QRS_NEXT_CUT()
PTP {E1 35817.199,E2 35817.199}
PTP {X 0,Y 759.903,A -85,B 0,C 180,E1 35817.199,E2 35817.199,E3 0,E4 0,E5 0,E6 0}
QRS_SPEED_INIT()
LIN {X 0,Y 759.903,Z 1215,A -85,B 0,C 180,E1 35817.199,E2 35817.199,E3 0,E4 0,E5 0,E6 0} C_VEL
LIN {X 0,Y 759.903,Z 294.644,A -85,B 0,C 180,E1 35817.199,E2 35817.199} C_VEL
LIN {X 0,Y 759.903,Z 286.569,A -85,B 0,C 180,E1 35817.199,E2 35817.199} C_VEL
LIN {X 0,Y 759.899,Z 284.569,A -85,B 0,C 180,E1 35817.048,E2 35817.048} C_VEL
LIN {X 0,Y 759.89,Z 284.574,A -85,B 0,C 180,E1 35814.261,E2 35814.261} C_VEL
LIN {X 0,Y 759.904,Z 284.564,A -85,B 0,C 180,E1 35811.373,E2 35811.373} C_VEL
LIN {X 0,Y 759.907,Z 284.576,A -85,B 0,C 180,E1 35808.309,E2 35808.309} C_VEL
LIN {X 0,Y 759.882,Z 284.567,A -85,B 0,C 180,E1 35805.444,E2 35805.444} C_VEL
LIN {X 0,Y 759.904,Z 284.571,A -85,B 0,C 180,E1 35802.621,E2 35802.621} C_VEL
LIN {X 0,Y 759.877,Z 284.573,A -85,B 0,C 180,E1 35799.833,E2 35799.833} C_VEL
LIN {X 0,Y 759.891,Z 284.566,A -85,B 0,C 180,E1 35797.077,E2 35797.077} C_VEL
LIN {X 0,Y 759.911,Z 284.577,A -85,B 0,C 180,E1 35794.097,E2 35794.097} C_VEL
LIN {X 0,Y 759.864,Z 284.571,A -85,B 0,C 180,E1 35791.362,E2 35791.362} C_VEL
LIN {X 0,Y 759.918,Z 284.564,A -85,B 0,C 180,E1 35788.597,E2 35788.597} C_VEL
LIN {X 0,Y 759.88,Z 284.575,A -85,B 0,C 180,E1 35785.632,E2 35785.632} C_VEL
LIN {X 0,Y 759.866,Z 284.568,A -85,B 0,C 180,E1 35782.938,E2 35782.938} C_VEL
LIN {X 0,Y 759.91,Z 284.572,A -85,B 0,C 180,E1 35780.093,E2 35780.093} C_VEL
LIN {X 0,Y 759.867,Z 284.574,A -85,B 0,C 180,E1 35777.337,E2 35777.337} C_VEL
LIN {X 0,Y 759.862,Z 284.57,A -85,B 0,C 180,E1 35774.718,E2 35774.718} C_VEL
LIN {X 0,Y 759.912,Z 284.571,A -85,B 0,C 180,E1 35771.944,E2 35771.944} C_VEL
LIN {X 0,Y 759.864,Z 284.575,A -85,B 0,C 180,E1 35769.168,E2 35769.168} C_VEL
LIN {X 0,Y 759.853,Z 284.57,A -85,B 0,C 180,E1 35766.59,E2 35766.59} C_VEL
LIN {X 0,Y 759.915,Z 284.571,A -85,B 0,C 180,E1 35763.818,E2 35763.818} C_VEL
LIN {X 0,Y 759.913,Z 284.828,A -85,B 0,C 180,E1 35761.644,E2 35761.644} C_VEL
LIN {X 0,Y 759.919,Z 312.056,A -85,B 0,C 180,E1 35759.876,E2 35759.876} C_VEL
LIN {X 0,Y 759.918,Z 346.9,A -85,B 0,C 180,E1 35757.717,E2 35757.717} C_VEL
LIN {X 0,Y 759.914,Z 568.445,A -85,B 0,C 180,E1 35755.191,E2 35755.191} C_VEL
LIN {X 0,Y 759.916,Z 778.609,A -85,B 0,C 180,E1 35752.849,E2 35752.849} C_VEL
LIN {X 0,Y 759.918,Z 798.366,A -85,B 0,C 180,E1 35752.545,E2 35752.545} C_VEL
LIN {X 0,Y 759.911,Z 822.306,A -85,B 0,C 180,E1 35752.064,E2 35752.064} C_VEL
LIN {X 0,Y 759.913,Z 846.929,A -85,B 0,C 180,E1 35751.415,E2 35751.415} C_VEL
LIN {X 0,Y 759.914,Z 866.189,A -85,B 0,C 180,E1 35750.809,E2 35750.809} C_VEL
LIN {X 0,Y 759.917,Z 885.052,A -85,B 0,C 180,E1 35750.125,E2 35750.125} C_VEL
LIN {X 0,Y 759.915,Z 904.461,A -85,B 0,C 180,E1 35749.324,E2 35749.324} C_VEL
LIN {X 0,Y 759.91,Z 928.8,A -85,B 0,C 180,E1 35748.17,E2 35748.17} C_VEL
LIN {X 0,Y 759.915,Z 948.392,A -85,B 0,C 180,E1 35747.102,E2 35747.102} C_VEL
LIN {X 0,Y 759.904,Z 967.176,A -85,B 0,C 180,E1 35745.962,E2 35745.962} C_VEL
LIN {X 0,Y 759.915,Z 988.802,A -85,B 0,C 180,E1 35744.477,E2 35744.477} C_VEL
LIN {X 0,Y 759.916,Z 1005.718,A -85,B 0,C 180,E1 35743.172,E2 35743.172} C_VEL
LIN {X 0,Y 759.903,Z 1024.655,A -85,B 0,C 180,E1 35741.537,E2 35741.537} C_VEL
LIN {X 0,Y 759.903,Z 1039.602,A -85,B 0,C 180,E1 35740.078,E2 35740.078} C_VEL
LIN {X 0,Y 759.901,Z 1054.389,A -85,B 0,C 180,E1 35738.474,E2 35738.474} C_VEL
LIN {X 0,Y 759.889,Z 1068.45,A -85,B 0,C 180,E1 35736.725,E2 35736.725} C_VEL
LIN {X 0,Y 759.91,Z 1079.205,A -85,B 0,C 180,E1 35735.209,E2 35735.209} C_VEL
LIN {X 0,Y 759.908,Z 1089.153,A -85,B 0,C 180,E1 35733.621,E2 35733.621} C_VEL
LIN {X 0,Y 759.901,Z 1099.607,A -85,B 0,C 180,E1 35731.659,E2 35731.659} C_VEL
LIN {X 0,Y 759.92,Z 1106.921,A -85,B 0,C 180,E1 35730,E2 35730} C_VEL
LIN {X 0,Y 759.904,Z 1112.724,A -85,B 0,C 180,E1 35728.417,E2 35728.417} C_VEL
LIN {X 0,Y 759.898,Z 1117.808,A -85,B 0,C 180,E1 35726.681,E2 35726.681} C_VEL
LIN {X 0,Y 759.903,Z 1121.967,A -85,B 0,C 180,E1 35724.64,E2 35724.64} C_VEL
LIN {X 0,Y 759.898,Z 1123.954,A -85,B 0,C 180,E1 35723.047,E2 35723.047} C_VEL
LIN {X 0,Y 759.902,Z 1124.86,A -85,B 0,C 180,E1 35721.449,E2 35721.449} C_VEL
LIN {X 0,Y 759.901,Z 1124.556,A -85,B 0,C 180,E1 35719.538,E2 35719.538} C_VEL
LIN {X 0,Y 759.916,Z 1122.598,A -85,B 0,C 180,E1 35717.693,E2 35717.693} C_VEL
LIN {X 0,Y 759.891,Z 1119.867,A -85,B 0,C 180,E1 35716.144,E2 35716.144} C_VEL
LIN {X 0,Y 759.916,Z 1116.057,A -85,B 0,C 180,E1 35714.587,E2 35714.587} C_VEL
LIN {X 0,Y 759.902,Z 1110.065,A -85,B 0,C 180,E1 35712.701,E2 35712.701} C_VEL
LIN {X 0,Y 759.909,Z 1102.135,A -85,B 0,C 180,E1 35710.796,E2 35710.796} C_VEL
LIN {X 0,Y 759.904,Z 1094.597,A -85,B 0,C 180,E1 35709.271,E2 35709.271} C_VEL
LIN {X 0,Y 759.901,Z 1085.453,A -85,B 0,C 180,E1 35707.672,E2 35707.672} C_VEL
LIN {X 0,Y 759.916,Z 1072.728,A -85,B 0,C 180,E1 35705.762,E2 35705.762} C_VEL
LIN {X 0,Y 759.909,Z 1060.564,A -85,B 0,C 180,E1 35704.182,E2 35704.182} C_VEL
LIN {X 0,Y 759.913,Z 1047.302,A -85,B 0,C 180,E1 35702.644,E2 35702.644} C_VEL
LIN {X 0,Y 759.908,Z 1029.889,A -85,B 0,C 180,E1 35700.867,E2 35700.867} C_VEL
LIN {X 0,Y 759.914,Z 1014.558,A -85,B 0,C 180,E1 35699.477,E2 35699.477} C_VEL
LIN {X 0,Y 759.914,Z 994.945,A -85,B 0,C 180,E1 35697.889,E2 35697.889} C_VEL
LIN {X 0,Y 759.9,Z 977.479,A -85,B 0,C 180,E1 35696.633,E2 35696.633} C_VEL
LIN {X 0,Y 759.915,Z 957.247,A -85,B 0,C 180,E1 35695.323,E2 35695.323} C_VEL
LIN {X 0,Y 759.914,Z 935.774,A -85,B 0,C 180,E1 35694.108,E2 35694.108} C_VEL
LIN {X 0,Y 759.912,Z 917.354,A -85,B 0,C 180,E1 35693.178,E2 35693.178} C_VEL
LIN {X 0,Y 759.915,Z 897.341,A -85,B 0,C 180,E1 35692.279,E2 35692.279} C_VEL
LIN {X 0,Y 759.918,Z 871.571,A -85,B 0,C 180,E1 35691.285,E2 35691.285} C_VEL
LIN {X 0,Y 759.915,Z 851.793,A -85,B 0,C 180,E1 35690.64,E2 35690.64} C_VEL
LIN {X 0,Y 759.916,Z 833.306,A -85,B 0,C 180,E1 35690.123,E2 35690.123} C_VEL
LIN {X 0,Y 759.913,Z 814.474,A -85,B 0,C 180,E1 35689.679,E2 35689.679} C_VEL
LIN {X 0,Y 759.912,Z 795.76,A -85,B 0,C 180,E1 35689.32,E2 35689.32} C_VEL
LIN {X 0,Y 759.913,Z 776.865,A -85,B 0,C 180,E1 35689.038,E2 35689.038} C_VEL
LIN {X 0,Y 759.915,Z 516.196,A -85,B 0,C 180,E1 35686.131,E2 35686.131} C_VEL
LIN {X 0,Y 759.913,Z 346.704,A -85,B 0,C 180,E1 35684.186,E2 35684.186} C_VEL
LIN {X 0,Y 759.917,Z 302.71,A -85,B 0,C 180,E1 35681.441,E2 35681.441} C_VEL
LIN {X 0,Y 759.904,Z 284.847,A -85,B 0,C 180,E1 35680.268,E2 35680.268} C_VEL
LIN {X 0,Y 759.912,Z 284.571,A -85,B 0,C 180,E1 35678.49,E2 35678.49} C_VEL
LIN {X 0,Y 759.917,Z 284.563,A -85,B 0,C 180,E1 35675.467,E2 35675.467} C_VEL
LIN {X 0,Y 759.891,Z 284.574,A -85,B 0,C 180,E1 35672.56,E2 35672.56} C_VEL
LIN {X 0,Y 759.894,Z 284.569,A -85,B 0,C 180,E1 35669.725,E2 35669.725} C_VEL
LIN {X 0,Y 759.894,Z 284.566,A -85,B 0,C 180,E1 35666.998,E2 35666.998} C_VEL
LIN {X 0,Y 759.912,Z 284.578,A -85,B 0,C 180,E1 35664.073,E2 35664.073} C_VEL
LIN {X 0,Y 759.916,Z 284.562,A -85,B 0,C 180,E1 35661.052,E2 35661.052} C_VEL
LIN {X 0,Y 759.911,Z 284.577,A -85,B 0,C 180,E1 35658.012,E2 35658.012} C_VEL
LIN {X 0,Y 759.909,Z 284.564,A -85,B 0,C 180,E1 35655.023,E2 35655.023} C_VEL
LIN {X 0,Y 759.891,Z 284.572,A -85,B 0,C 180,E1 35652.141,E2 35652.141} C_VEL
LIN {X 0,Y 759.894,Z 284.572,A -85,B 0,C 180,E1 35649.391,E2 35649.391} C_VEL
LIN {X 0,Y 759.908,Z 284.563,A -85,B 0,C 180,E1 35646.573,E2 35646.573} C_VEL
LIN {X 0,Y 759.915,Z 284.577,A -85,B 0,C 180,E1 35643.621,E2 35643.621} C_VEL
LIN {X 0,Y 759.907,Z 284.563,A -85,B 0,C 180,E1 35640.603,E2 35640.603} C_VEL
LIN {X 0,Y 759.9,Z 284.574,A -85,B 0,C 180,E1 35637.662,E2 35637.662} C_VEL
LIN {X 0,Y 759.888,Z 284.57,A -85,B 0,C 180,E1 35634.866,E2 35634.866} C_VEL
LIN {X 0,Y 759.9,Z 284.566,A -85,B 0,C 180,E1 35632.059,E2 35632.059} C_VEL
LIN {X 0,Y 759.909,Z 284.576,A -85,B 0,C 180,E1 35629.155,E2 35629.155} C_VEL
LIN {X 0,Y 759.911,Z 284.563,A -85,B 0,C 180,E1 35626.144,E2 35626.144} C_VEL
LIN {X 0,Y 759.919,Z 284.577,A -85,B 0,C 180,E1 35623.095,E2 35623.095} C_VEL
LIN {X 0,Y 759.905,Z 284.563,A -85,B 0,C 180,E1 35620.075,E2 35620.075} C_VEL
LIN {X 0,Y 759.909,Z 284.576,A -85,B 0,C 180,E1 35617.077,E2 35617.077} C_VEL
LIN {X 0,Y 759.883,Z 284.569,A -85,B 0,C 180,E1 35614.264,E2 35614.264} C_VEL
LIN {X 0,Y 759.901,Z 284.566,A -85,B 0,C 180,E1 35611.468,E2 35611.468} C_VEL
LIN {X 0,Y 759.901,Z 284.576,A -85,B 0,C 180,E1 35608.596,E2 35608.596} C_VEL
LIN {X 0,Y 759.899,Z 284.565,A -85,B 0,C 180,E1 35605.721,E2 35605.721} C_VEL
LIN {X 0,Y 759.902,Z 284.574,A -85,B 0,C 180,E1 35602.846,E2 35602.846} C_VEL
LIN {X 0,Y 759.879,Z 284.572,A -85,B 0,C 180,E1 35600.048,E2 35600.048} C_VEL
LIN {X 0,Y 759.91,Z 284.562,A -85,B 0,C 180,E1 35597.238,E2 35597.238} C_VEL
LIN {X 0,Y 759.902,Z 284.796,A -85,B 0,C 180,E1 35594.679,E2 35594.679} C_VEL
LIN {X 0,Y 759.918,Z 288.931,A -85,B 0,C 180,E1 35594.4,E2 35594.4} C_VEL
LIN {X 0,Y 759.896,Z 333.48,A -85,B 0,C 180,E1 35591.844,E2 35591.844} C_VEL
LIN {X 0,Y 759.909,Z 350.22,A -85,B 0,C 180,E1 35590.926,E2 35590.926} C_VEL
LIN {X 0,Y 759.918,Z 558.925,A -85,B 0,C 180,E1 35588.412,E2 35588.412} C_VEL
LIN {X 0,Y 759.917,Z 786.633,A -85,B 0,C 180,E1 35585.769,E2 35585.769} C_VEL
LIN {X 0,Y 759.91,Z 830.472,A -85,B 0,C 180,E1 35585.243,E2 35585.243} C_VEL
LIN {X 0,Y 759.91,Z 856.594,A -85,B 0,C 180,E1 35584.789,E2 35584.789} C_VEL
LIN {X 0,Y 759.914,Z 883.601,A -85,B 0,C 180,E1 35584.163,E2 35584.163} C_VEL
LIN {X 0,Y 759.908,Z 907.506,A -85,B 0,C 180,E1 35583.465,E2 35583.465} C_VEL
LIN {X 0,Y 759.918,Z 931.763,A -85,B 0,C 180,E1 35582.637,E2 35582.637} C_VEL
LIN {X 0,Y 759.917,Z 956.965,A -85,B 0,C 180,E1 35581.611,E2 35581.611} C_VEL
LIN {X 0,Y 759.912,Z 976.742,A -85,B 0,C 180,E1 35580.698,E2 35580.698} C_VEL
LIN {X 0,Y 759.913,Z 995.424,A -85,B 0,C 180,E1 35579.738,E2 35579.738} C_VEL
LIN {X 0,Y 759.909,Z 1013.705,A -85,B 0,C 180,E1 35578.702,E2 35578.702} C_VEL
LIN {X 0,Y 759.911,Z 1035.513,A -85,B 0,C 180,E1 35577.335,E2 35577.335} C_VEL
LIN {X 0,Y 759.912,Z 1056.843,A -85,B 0,C 180,E1 35575.818,E2 35575.818} C_VEL
LIN {X 0,Y 759.91,Z 1073.821,A -85,B 0,C 180,E1 35574.486,E2 35574.486} C_VEL
LIN {X 0,Y 759.901,Z 1092.852,A -85,B 0,C 180,E1 35572.84,E2 35572.84} C_VEL
LIN {X 0,Y 759.895,Z 1109.493,A -85,B 0,C 180,E1 35571.213,E2 35571.213} C_VEL
LIN {X 0,Y 759.905,Z 1122.957,A -85,B 0,C 180,E1 35569.764,E2 35569.764} C_VEL
LIN {X 0,Y 759.897,Z 1135.731,A -85,B 0,C 180,E1 35568.25,E2 35568.25} C_VEL
LIN {X 0,Y 759.909,Z 1150.031,A -85,B 0,C 180,E1 35566.354,E2 35566.354} C_VEL
LIN {X 0,Y 759.909,Z 1162.194,A -85,B 0,C 180,E1 35564.477,E2 35564.477} C_VEL
LIN {X 0,Y 759.91,Z 1171.058,A -85,B 0,C 180,E1 35562.925,E2 35562.925} C_VEL
LIN {X 0,Y 759.91,Z 1178.784,A -85,B 0,C 180,E1 35561.383,E2 35561.383} C_VEL
LIN {X 0,Y 759.906,Z 1186.43,A -85,B 0,C 180,E1 35559.619,E2 35559.619} C_VEL
LIN {X 0,Y 759.908,Z 1193.594,A -85,B 0,C 180,E1 35557.561,E2 35557.561} C_VEL
LIN {X 0,Y 759.91,Z 1199.108,A -85,B 0,C 180,E1 35555.436,E2 35555.436} C_VEL
LIN {X 0,Y 759.916,Z 1202.585,A -85,B 0,C 180,E1 35553.47,E2 35553.47} C_VEL
LIN {X 0,Y 759.914,Z 1204.58,A -85,B 0,C 180,E1 35551.433,E2 35551.433} C_VEL
LIN {X 0,Y 759.889,Z 1204.849,A -85,B 0,C 180,E1 35549.472,E2 35549.472} C_VEL
LIN {X 0,Y 759.907,Z 1203.907,A -85,B 0,C 180,E1 35547.662,E2 35547.662} C_VEL
LIN {X 0,Y 759.908,Z 1201.054,A -85,B 0,C 180,E1 35545.548,E2 35545.548} C_VEL
LIN {X 0,Y 759.914,Z 1196.566,A -85,B 0,C 180,E1 35543.503,E2 35543.503} C_VEL
LIN {X 0,Y 759.912,Z 1190.629,A -85,B 0,C 180,E1 35541.526,E2 35541.526} C_VEL
LIN {X 0,Y 759.896,Z 1182.681,A -85,B 0,C 180,E1 35539.462,E2 35539.462} C_VEL
LIN {X 0,Y 759.905,Z 1173.111,A -85,B 0,C 180,E1 35537.461,E2 35537.461} C_VEL
LIN {X 0,Y 759.91,Z 1164.056,A -85,B 0,C 180,E1 35535.834,E2 35535.834} C_VEL
LIN {X 0,Y 759.894,Z 1154.212,A -85,B 0,C 180,E1 35534.273,E2 35534.273} C_VEL
LIN {X 0,Y 759.904,Z 1143.666,A -85,B 0,C 180,E1 35532.78,E2 35532.78} C_VEL
LIN {X 0,Y 759.896,Z 1130.456,A -85,B 0,C 180,E1 35531.1,E2 35531.1} C_VEL
LIN {X 0,Y 759.898,Z 1113.394,A -85,B 0,C 180,E1 35529.191,E2 35529.191} C_VEL
LIN {X 0,Y 759.898,Z 1098.828,A -85,B 0,C 180,E1 35527.732,E2 35527.732} C_VEL
LIN {X 0,Y 759.911,Z 1082.654,A -85,B 0,C 180,E1 35526.258,E2 35526.258} C_VEL
LIN {X 0,Y 759.91,Z 1061.274,A -85,B 0,C 180,E1 35524.516,E2 35524.516} C_VEL
LIN {X 0,Y 759.91,Z 1044.049,A -85,B 0,C 180,E1 35523.257,E2 35523.257} C_VEL
LIN {X 0,Y 759.914,Z 1026.242,A -85,B 0,C 180,E1 35522.069,E2 35522.069} C_VEL
LIN {X 0,Y 759.905,Z 1003.453,A -85,B 0,C 180,E1 35520.695,E2 35520.695} C_VEL
LIN {X 0,Y 759.916,Z 981.266,A -85,B 0,C 180,E1 35519.525,E2 35519.525} C_VEL
LIN {X 0,Y 759.912,Z 961.681,A -85,B 0,C 180,E1 35518.598,E2 35518.598} C_VEL
LIN {X 0,Y 759.918,Z 942.461,A -85,B 0,C 180,E1 35517.785,E2 35517.785} C_VEL
LIN {X 0,Y 759.919,Z 923.852,A -85,B 0,C 180,E1 35517.085,E2 35517.085} C_VEL
LIN {X 0,Y 759.909,Z 905.509,A -85,B 0,C 180,E1 35516.474,E2 35516.474} C_VEL
LIN {X 0,Y 759.914,Z 882.834,A -85,B 0,C 180,E1 35515.818,E2 35515.818} C_VEL
LIN {X 0,Y 759.911,Z 855.669,A -85,B 0,C 180,E1 35515.191,E2 35515.191} C_VEL
LIN {X 0,Y 759.909,Z 829.102,A -85,B 0,C 180,E1 35514.737,E2 35514.737} C_VEL
LIN {X 0,Y 759.918,Z 735.97,A -85,B 0,C 180,E1 35513.651,E2 35513.651} C_VEL
LIN {X 0,Y 759.915,Z 513.131,A -85,B 0,C 180,E1 35511.045,E2 35511.045} C_VEL
LIN {X 0,Y 759.909,Z 349.756,A -85,B 0,C 180,E1 35509.062,E2 35509.062} C_VEL
LIN {X 0,Y 759.917,Z 304.694,A -85,B 0,C 180,E1 35506.517,E2 35506.517} C_VEL
LIN {X 0,Y 759.903,Z 284.954,A -85,B 0,C 180,E1 35505.342,E2 35505.342} C_VEL
LIN {X 0,Y 759.905,Z 284.552,A -85,B 0,C 180,E1 35504.937,E2 35504.937} C_VEL
LIN {X 0,Y 759.88,Z 284.567,A -85,B 0,C 180,E1 35502.151,E2 35502.151} C_VEL
LIN {X 0,Y 759.906,Z 284.575,A -85,B 0,C 180,E1 35499.316,E2 35499.316} C_VEL
LIN {X 0,Y 759.903,Z 284.564,A -85,B 0,C 180,E1 35496.366,E2 35496.366} C_VEL
LIN {X 0,Y 759.915,Z 284.577,A -85,B 0,C 180,E1 35493.367,E2 35493.367} C_VEL
LIN {X 0,Y 759.914,Z 284.563,A -85,B 0,C 180,E1 35490.33,E2 35490.33} C_VEL
LIN {X 0,Y 759.905,Z 284.576,A -85,B 0,C 180,E1 35487.337,E2 35487.337} C_VEL
LIN {X 0,Y 759.9,Z 284.566,A -85,B 0,C 180,E1 35484.404,E2 35484.404} C_VEL
LIN {X 0,Y 759.889,Z 284.569,A -85,B 0,C 180,E1 35481.619,E2 35481.619} C_VEL
LIN {X 0,Y 759.899,Z 284.574,A -85,B 0,C 180,E1 35478.807,E2 35478.807} C_VEL
LIN {X 0,Y 759.912,Z 284.562,A -85,B 0,C 180,E1 35475.884,E2 35475.884} C_VEL
LIN {X 0,Y 759.909,Z 284.577,A -85,B 0,C 180,E1 35472.845,E2 35472.845} C_VEL
LIN {X 0,Y 759.911,Z 284.562,A -85,B 0,C 180,E1 35469.849,E2 35469.849} C_VEL
LIN {X 0,Y 759.917,Z 284.577,A -85,B 0,C 180,E1 35466.801,E2 35466.801} C_VEL
LIN {X 0,Y 759.889,Z 284.567,A -85,B 0,C 180,E1 35463.923,E2 35463.923} C_VEL
LIN {X 0,Y 759.897,Z 284.569,A -85,B 0,C 180,E1 35461.131,E2 35461.131} C_VEL
LIN {X 0,Y 759.891,Z 284.574,A -85,B 0,C 180,E1 35458.341,E2 35458.341} C_VEL
LIN {X 0,Y 759.899,Z 284.569,A -85,B 0,C 180,E1 35457.048,E2 35457.048} C_VEL
LIN {X 0,Y 758.92,Z 284.701,A -85,B 0,C 180,E1 35456.467,E2 35456.467} C_VEL
LIN {X 0,Y 752.526,Z 285.503,A -85,B 0,C 180,E1 35454.841,E2 35454.841} C_VEL
LIN {X 0,Y 751.966,Z 285.565,A -85,B 0,C 180,E1 35454.418,E2 35454.418} C_VEL
LIN {X 0,Y 751.952,Z 285.555,A -85,B 0,C 180,E1 35451.512,E2 35451.512} C_VEL
LIN {X 0,Y 751.969,Z 285.563,A -85,B 0,C 180,E1 35448.573,E2 35448.573} C_VEL
LIN {X 0,Y 751.935,Z 285.56,A -85,B 0,C 180,E1 35445.759,E2 35445.759} C_VEL
LIN {X 0,Y 751.974,Z 285.553,A -85,B 0,C 180,E1 35442.943,E2 35442.943} C_VEL
LIN {X 0,Y 751.953,Z 285.564,A -85,B 0,C 180,E1 35440.017,E2 35440.017} C_VEL
LIN {X 0,Y 751.939,Z 285.557,A -85,B 0,C 180,E1 35437.235,E2 35437.235} C_VEL
LIN {X 0,Y 751.97,Z 285.559,A -85,B 0,C 180,E1 35434.311,E2 35434.311} C_VEL
LIN {X 0,Y 751.929,Z 285.561,A -85,B 0,C 180,E1 35431.515,E2 35431.515} C_VEL
LIN {X 0,Y 751.962,Z 285.552,A -85,B 0,C 180,E1 35428.757,E2 35428.757} C_VEL
LIN {X 0,Y 751.956,Z 285.565,A -85,B 0,C 180,E1 35425.773,E2 35425.773} C_VEL
LIN {X 0,Y 751.923,Z 285.556,A -85,B 0,C 180,E1 35423.051,E2 35423.051} C_VEL
LIN {X 0,Y 751.974,Z 285.558,A -85,B 0,C 180,E1 35420.239,E2 35420.239} C_VEL
LIN {X 0,Y 751.934,Z 285.563,A -85,B 0,C 180,E1 35417.402,E2 35417.402} C_VEL
LIN {X 0,Y 751.921,Z 285.559,A -85,B 0,C 180,E1 35414.756,E2 35414.756} C_VEL
LIN {X 0,Y 751.974,Z 285.559,A -85,B 0,C 180,E1 35411.975,E2 35411.975} C_VEL
LIN {X 0,Y 751.925,Z 285.564,A -85,B 0,C 180,E1 35409.17,E2 35409.17} C_VEL
LIN {X 0,Y 751.916,Z 285.559,A -85,B 0,C 180,E1 35406.563,E2 35406.563} C_VEL
LIN {X 0,Y 751.976,Z 285.563,A -85,B 0,C 180,E1 35403.765,E2 35403.765} C_VEL
LIN {X 0,Y 751.975,Z 285.761,A -85,B 0,C 180,E1 35402.112,E2 35402.112} C_VEL
LIN {X 0,Y 753.211,Z 289.399,A -85,B 0,C 180,E1 35401.758,E2 35401.758} C_VEL
LIN {X 0,Y 753.045,Z 330.759,A -85,B 0,C 180,E1 35399.109,E2 35399.109} C_VEL
LIN {X 0,Y 753.126,Z 347.248,A -85,B 0,C 180,E1 35398.098,E2 35398.098} C_VEL
LIN {X 0,Y 753.494,Z 350.648,A -85,B 0,C 180,E1 35398.032,E2 35398.032} C_VEL
LIN {X 0,Y 753.268,Z 592.033,A -85,B 0,C 180,E1 35395.269,E2 35395.269} C_VEL
LIN {X 0,Y 753.108,Z 779.265,A -85,B 0,C 180,E1 35393.163,E2 35393.163} C_VEL
LIN {X 0,Y 753.068,Z 800.182,A -85,B 0,C 180,E1 35392.835,E2 35392.835} C_VEL
LIN {X 0,Y 752.971,Z 826.736,A -85,B 0,C 180,E1 35392.273,E2 35392.273} C_VEL
LIN {X 0,Y 752.903,Z 848.373,A -85,B 0,C 180,E1 35391.686,E2 35391.686} C_VEL
LIN {X 0,Y 752.833,Z 868.046,A -85,B 0,C 180,E1 35391.055,E2 35391.055} C_VEL
LIN {X 0,Y 752.755,Z 888.779,A -85,B 0,C 180,E1 35390.284,E2 35390.284} C_VEL
LIN {X 0,Y 752.626,Z 913.899,A -85,B 0,C 180,E1 35389.192,E2 35389.192} C_VEL
LIN {X 0,Y 752.536,Z 933.823,A -85,B 0,C 180,E1 35388.191,E2 35388.191} C_VEL
LIN {X 0,Y 752.446,Z 954.28,A -85,B 0,C 180,E1 35387.038,E2 35387.038} C_VEL
LIN {X 0,Y 752.334,Z 975.831,A -85,B 0,C 180,E1 35385.652,E2 35385.652} C_VEL
LIN {X 0,Y 752.271,Z 993.317,A -85,B 0,C 180,E1 35384.391,E2 35384.391} C_VEL
LIN {X 0,Y 752.161,Z 1013.62,A -85,B 0,C 180,E1 35382.748,E2 35382.748} C_VEL
LIN {X 0,Y 752.119,Z 1028.977,A -85,B 0,C 180,E1 35381.347,E2 35381.347} C_VEL
LIN {X 0,Y 752.047,Z 1045.726,A -85,B 0,C 180,E1 35379.644,E2 35379.644} C_VEL
LIN {X 0,Y 751.999,Z 1059.636,A -85,B 0,C 180,E1 35378.025,E2 35378.025} C_VEL
LIN {X 0,Y 751.966,Z 1070.868,A -85,B 0,C 180,E1 35376.566,E2 35376.566} C_VEL
LIN {X 0,Y 751.958,Z 1082.901,A -85,B 0,C 180,E1 35374.805,E2 35374.805} C_VEL
LIN {X 0,Y 751.93,Z 1093.527,A -85,B 0,C 180,E1 35372.968,E2 35372.968} C_VEL
LIN {X 0,Y 751.925,Z 1101.455,A -85,B 0,C 180,E1 35371.371,E2 35371.371} C_VEL
LIN {X 0,Y 751.906,Z 1108.209,A -85,B 0,C 180,E1 35369.771,E2 35369.771} C_VEL
LIN {X 0,Y 751.916,Z 1114.983,A -85,B 0,C 180,E1 35367.79,E2 35367.79} C_VEL
LIN {X 0,Y 751.919,Z 1119.571,A -85,B 0,C 180,E1 35365.959,E2 35365.959} C_VEL
LIN {X 0,Y 751.892,Z 1122.449,A -85,B 0,C 180,E1 35364.353,E2 35364.353} C_VEL
LIN {X 0,Y 751.906,Z 1124.31,A -85,B 0,C 180,E1 35362.666,E2 35362.666} C_VEL
LIN {X 0,Y 751.904,Z 1124.898,A -85,B 0,C 180,E1 35360.586,E2 35360.586} C_VEL
LIN {X 0,Y 751.901,Z 1123.992,A -85,B 0,C 180,E1 35358.883,E2 35358.883} C_VEL
LIN {X 0,Y 751.913,Z 1121.991,A -85,B 0,C 180,E1 35357.248,E2 35357.248} C_VEL
LIN {X 0,Y 751.896,Z 1118.128,A -85,B 0,C 180,E1 35355.286,E2 35355.286} C_VEL
LIN {X 0,Y 751.92,Z 1112.901,A -85,B 0,C 180,E1 35353.467,E2 35353.467} C_VEL
LIN {X 0,Y 751.925,Z 1107.15,A -85,B 0,C 180,E1 35351.871,E2 35351.871} C_VEL
LIN {X 0,Y 751.912,Z 1099.803,A -85,B 0,C 180,E1 35350.179,E2 35350.179} C_VEL
LIN {X 0,Y 751.949,Z 1089.088,A -85,B 0,C 180,E1 35348.142,E2 35348.142} C_VEL
LIN {X 0,Y 751.951,Z 1079.331,A -85,B 0,C 180,E1 35346.566,E2 35346.566} C_VEL
LIN {X 0,Y 751.985,Z 1068.249,A -85,B 0,C 180,E1 35344.987,E2 35344.987} C_VEL
LIN {X 0,Y 752.039,Z 1053.317,A -85,B 0,C 180,E1 35343.125,E2 35343.125} C_VEL
LIN {X 0,Y 752.075,Z 1039.161,A -85,B 0,C 180,E1 35341.579,E2 35341.579} C_VEL
LIN {X 0,Y 752.137,Z 1023.19,A -85,B 0,C 180,E1 35340.011,E2 35340.011} C_VEL
LIN {X 0,Y 752.207,Z 1004.978,A -85,B 0,C 180,E1 35338.438,E2 35338.438} C_VEL
LIN {X 0,Y 752.277,Z 987.356,A -85,B 0,C 180,E1 35337.071,E2 35337.071} C_VEL
LIN {X 0,Y 752.383,Z 966.1,A -85,B 0,C 180,E1 35335.612,E2 35335.612} C_VEL
LIN {X 0,Y 752.47,Z 947.046,A -85,B 0,C 180,E1 35334.451,E2 35334.451} C_VEL
LIN {X 0,Y 752.599,Z 924.683,A -85,B 0,C 180,E1 35333.239,E2 35333.239} C_VEL
LIN {X 0,Y 752.686,Z 903.01,A -85,B 0,C 180,E1 35332.225,E2 35332.225} C_VEL
LIN {X 0,Y 752.767,Z 883.493,A -85,B 0,C 180,E1 35331.42,E2 35331.42} C_VEL
LIN {X 0,Y 752.852,Z 861.286,A -85,B 0,C 180,E1 35330.622,E2 35330.622} C_VEL
LIN {X 0,Y 752.959,Z 835.793,A -85,B 0,C 180,E1 35329.87,E2 35329.87} C_VEL
LIN {X 0,Y 753.018,Z 815.115,A -85,B 0,C 180,E1 35329.374,E2 35329.374} C_VEL
LIN {X 0,Y 753.067,Z 795.379,A -85,B 0,C 180,E1 35328.992,E2 35328.992} C_VEL
LIN {X 0,Y 753.109,Z 775.7,A -85,B 0,C 180,E1 35328.7,E2 35328.7} C_VEL
LIN {X 0,Y 753.337,Z 518.031,A -85,B 0,C 180,E1 35325.804,E2 35325.804} C_VEL
LIN {X 0,Y 753.318,Z 348.126,A -85,B 0,C 180,E1 35323.837,E2 35323.837} C_VEL
LIN {X 0,Y 753.006,Z 345.56,A -85,B 0,C 180,E1 35323.727,E2 35323.727} C_VEL
LIN {X 0,Y 753.167,Z 302.195,A -85,B 0,C 180,E1 35320.983,E2 35320.983} C_VEL
LIN {X 0,Y 753.023,Z 288.662,A -85,B 0,C 180,E1 35320.091,E2 35320.091} C_VEL
LIN {X 0,Y 751.984,Z 285.677,A -85,B 0,C 180,E1 35319.778,E2 35319.778} C_VEL
LIN {X 0,Y 751.942,Z 285.562,A -85,B 0,C 180,E1 35316.945,E2 35316.945} C_VEL
LIN {X 0,Y 751.966,Z 285.565,A -85,B 0,C 180,E1 35314.134,E2 35314.134} C_VEL
LIN {X 0,Y 751.966,Z 285.554,A -85,B 0,C 180,E1 35311.237,E2 35311.237} C_VEL
LIN {X 0,Y 751.97,Z 285.564,A -85,B 0,C 180,E1 35308.254,E2 35308.254} C_VEL
LIN {X 0,Y 751.974,Z 285.551,A -85,B 0,C 180,E1 35305.182,E2 35305.182} C_VEL
LIN {X 0,Y 751.965,Z 285.565,A -85,B 0,C 180,E1 35302.187,E2 35302.187} C_VEL
LIN {X 0,Y 751.963,Z 285.555,A -85,B 0,C 180,E1 35299.255,E2 35299.255} C_VEL
LIN {X 0,Y 751.947,Z 285.556,A -85,B 0,C 180,E1 35296.453,E2 35296.453} C_VEL
LIN {X 0,Y 751.962,Z 285.561,A -85,B 0,C 180,E1 35293.613,E2 35293.613} C_VEL
LIN {X 0,Y 751.97,Z 285.552,A -85,B 0,C 180,E1 35290.7,E2 35290.7} C_VEL
LIN {X 0,Y 751.971,Z 285.564,A -85,B 0,C 180,E1 35287.718,E2 35287.718} C_VEL
LIN {X 0,Y 751.976,Z 285.552,A -85,B 0,C 180,E1 35284.652,E2 35284.652} C_VEL
LIN {X 0,Y 751.97,Z 285.564,A -85,B 0,C 180,E1 35281.6,E2 35281.6} C_VEL
LIN {X 0,Y 751.965,Z 285.554,A -85,B 0,C 180,E1 35278.629,E2 35278.629} C_VEL
LIN {X 0,Y 751.955,Z 285.559,A -85,B 0,C 180,E1 35275.73,E2 35275.73} C_VEL
LIN {X 0,Y 751.951,Z 285.561,A -85,B 0,C 180,E1 35272.973,E2 35272.973} C_VEL
LIN {X 0,Y 751.97,Z 285.55,A -85,B 0,C 180,E1 35270.123,E2 35270.123} C_VEL
LIN {X 0,Y 751.976,Z 285.565,A -85,B 0,C 180,E1 35267.17,E2 35267.17} C_VEL
LIN {X 0,Y 751.968,Z 285.552,A -85,B 0,C 180,E1 35264.182,E2 35264.182} C_VEL
LIN {X 0,Y 751.966,Z 285.564,A -85,B 0,C 180,E1 35261.212,E2 35261.212} C_VEL
LIN {X 0,Y 751.947,Z 285.558,A -85,B 0,C 180,E1 35258.35,E2 35258.35} C_VEL
LIN {X 0,Y 751.961,Z 285.553,A -85,B 0,C 180,E1 35255.572,E2 35255.572} C_VEL
LIN {X 0,Y 751.959,Z 285.562,A -85,B 0,C 180,E1 35252.65,E2 35252.65} C_VEL
LIN {X 0,Y 751.971,Z 285.553,A -85,B 0,C 180,E1 35249.738,E2 35249.738} C_VEL
LIN {X 0,Y 751.972,Z 285.566,A -85,B 0,C 180,E1 35246.69,E2 35246.69} C_VEL
LIN {X 0,Y 751.949,Z 285.557,A -85,B 0,C 180,E1 35243.814,E2 35243.814} C_VEL
LIN {X 0,Y 751.96,Z 285.56,A -85,B 0,C 180,E1 35241.027,E2 35241.027} C_VEL
LIN {X 0,Y 751.95,Z 285.557,A -85,B 0,C 180,E1 35238.226,E2 35238.226} C_VEL
LIN {X 0,Y 751.983,Z 285.616,A -85,B 0,C 180,E1 35235.3,E2 35235.3} C_VEL
LIN {X 0,Y 752.13,Z 286.411,A -85,B 0,C 180,E1 35235.142,E2 35235.142} C_VEL
LIN {X 0,Y 753.598,Z 289.622,A -85,B 0,C 180,E1 35234.831,E2 35234.831} C_VEL
LIN {X 0,Y 753.424,Z 332.615,A -85,B 0,C 180,E1 35232.335,E2 35232.335} C_VEL
LIN {X 0,Y 753.504,Z 350.421,A -85,B 0,C 180,E1 35231.346,E2 35231.346} C_VEL
LIN {X 0,Y 753.844,Z 353.801,A -85,B 0,C 180,E1 35231.279,E2 35231.279} C_VEL
LIN {X 0,Y 753.627,Z 565.931,A -85,B 0,C 180,E1 35228.708,E2 35228.708} C_VEL
LIN {X 0,Y 753.41,Z 792.333,A -85,B 0,C 180,E1 35226.061,E2 35226.061} C_VEL
LIN {X 0,Y 753.349,Z 832.416,A -85,B 0,C 180,E1 35225.568,E2 35225.568} C_VEL
LIN {X 0,Y 753.272,Z 858.587,A -85,B 0,C 180,E1 35225.098,E2 35225.098} C_VEL
LIN {X 0,Y 753.187,Z 885.146,A -85,B 0,C 180,E1 35224.469,E2 35224.469} C_VEL
LIN {X 0,Y 753.089,Z 911.441,A -85,B 0,C 180,E1 35223.686,E2 35223.686} C_VEL
LIN {X 0,Y 752.955,Z 937.244,A -85,B 0,C 180,E1 35222.76,E2 35222.76} C_VEL
LIN {X 0,Y 752.856,Z 958.7,A -85,B 0,C 180,E1 35221.865,E2 35221.865} C_VEL
LIN {X 0,Y 752.759,Z 977.635,A -85,B 0,C 180,E1 35220.977,E2 35220.977} C_VEL
LIN {X 0,Y 752.665,Z 996.704,A -85,B 0,C 180,E1 35219.984,E2 35219.984} C_VEL
LIN {X 0,Y 752.56,Z 1016.618,A -85,B 0,C 180,E1 35218.835,E2 35218.835} C_VEL
LIN {X 0,Y 752.413,Z 1040.42,A -85,B 0,C 180,E1 35217.288,E2 35217.288} C_VEL
LIN {X 0,Y 752.343,Z 1058.504,A -85,B 0,C 180,E1 35215.97,E2 35215.97} C_VEL
LIN {X 0,Y 752.263,Z 1076.36,A -85,B 0,C 180,E1 35214.542,E2 35214.542} C_VEL
LIN {X 0,Y 752.17,Z 1096.267,A -85,B 0,C 180,E1 35212.757,E2 35212.757} C_VEL
LIN {X 0,Y 752.095,Z 1111.284,A -85,B 0,C 180,E1 35211.257,E2 35211.257} C_VEL
LIN {X 0,Y 752.063,Z 1125.174,A -85,B 0,C 180,E1 35209.727,E2 35209.727} C_VEL
LIN {X 0,Y 752.008,Z 1141.338,A -85,B 0,C 180,E1 35207.727,E2 35207.727} C_VEL
LIN {X 0,Y 751.956,Z 1153.167,A -85,B 0,C 180,E1 35206.056,E2 35206.056} C_VEL
LIN {X 0,Y 751.955,Z 1163.126,A -85,B 0,C 180,E1 35204.476,E2 35204.476} C_VEL
LIN {X 0,Y 751.94,Z 1171.88,A -85,B 0,C 180,E1 35202.908,E2 35202.908} C_VEL
LIN {X 0,Y 751.93,Z 1179.5,A -85,B 0,C 180,E1 35201.35,E2 35201.35} C_VEL
LIN {X 0,Y 751.916,Z 1187.31,A -85,B 0,C 180,E1 35199.491,E2 35199.491} C_VEL
LIN {X 0,Y 751.911,Z 1194.033,A -85,B 0,C 180,E1 35197.488,E2 35197.488} C_VEL
LIN {X 0,Y 751.911,Z 1199.28,A -85,B 0,C 180,E1 35195.418,E2 35195.418} C_VEL
LIN {X 0,Y 751.914,Z 1202.789,A -85,B 0,C 180,E1 35193.354,E2 35193.354} C_VEL
LIN {X 0,Y 751.915,Z 1204.603,A -85,B 0,C 180,E1 35191.372,E2 35191.372} C_VEL
LIN {X 0,Y 751.889,Z 1204.849,A -85,B 0,C 180,E1 35189.467,E2 35189.467} C_VEL
LIN {X 0,Y 751.907,Z 1203.907,A -85,B 0,C 180,E1 35187.638,E2 35187.638} C_VEL
LIN {X 0,Y 751.907,Z 1201.054,A -85,B 0,C 180,E1 35185.5,E2 35185.5} C_VEL
LIN {X 0,Y 751.912,Z 1196.566,A -85,B 0,C 180,E1 35183.433,E2 35183.433} C_VEL
LIN {X 0,Y 751.92,Z 1190.63,A -85,B 0,C 180,E1 35181.435,E2 35181.435} C_VEL
LIN {X 0,Y 751.905,Z 1182.636,A -85,B 0,C 180,E1 35179.338,E2 35179.338} C_VEL
LIN {X 0,Y 751.935,Z 1173.112,A -85,B 0,C 180,E1 35177.326,E2 35177.326} C_VEL
LIN {X 0,Y 751.955,Z 1164.058,A -85,B 0,C 180,E1 35175.681,E2 35175.681} C_VEL
LIN {X 0,Y 751.954,Z 1154.214,A -85,B 0,C 180,E1 35174.103,E2 35174.103} C_VEL
LIN {X 0,Y 752.006,Z 1143.086,A -85,B 0,C 180,E1 35172.513,E2 35172.513} C_VEL
LIN {X 0,Y 752.065,Z 1127.932,A -85,B 0,C 180,E1 35170.587,E2 35170.587} C_VEL
LIN {X 0,Y 752.088,Z 1112.616,A -85,B 0,C 180,E1 35168.883,E2 35168.883} C_VEL
LIN {X 0,Y 752.166,Z 1097.976,A -85,B 0,C 180,E1 35167.408,E2 35167.408} C_VEL
LIN {X 0,Y 752.232,Z 1079.86,A -85,B 0,C 180,E1 35165.75,E2 35165.75} C_VEL
LIN {X 0,Y 752.347,Z 1060.167,A -85,B 0,C 180,E1 35164.157,E2 35164.157} C_VEL
LIN {X 0,Y 752.409,Z 1042.84,A -85,B 0,C 180,E1 35162.883,E2 35162.883} C_VEL
LIN {X 0,Y 752.521,Z 1022.27,A -85,B 0,C 180,E1 35161.511,E2 35161.511} C_VEL
LIN {X 0,Y 752.657,Z 998.639,A -85,B 0,C 180,E1 35160.122,E2 35160.122} C_VEL
LIN {X 0,Y 752.754,Z 979.254,A -85,B 0,C 180,E1 35159.103,E2 35159.103} C_VEL
LIN {X 0,Y 752.851,Z 960.434,A -85,B 0,C 180,E1 35158.213,E2 35158.213} C_VEL
LIN {X 0,Y 752.948,Z 940.603,A -85,B 0,C 180,E1 35157.375,E2 35157.375} C_VEL
LIN {X 0,Y 753.037,Z 920.043,A -85,B 0,C 180,E1 35156.608,E2 35156.608} C_VEL
LIN {X 0,Y 753.159,Z 894.912,A -85,B 0,C 180,E1 35155.802,E2 35155.802} C_VEL
LIN {X 0,Y 753.243,Z 867.448,A -85,B 0,C 180,E1 35155.094,E2 35155.094} C_VEL
LIN {X 0,Y 753.329,Z 841.929,A -85,B 0,C 180,E1 35154.586,E2 35154.586} C_VEL
LIN {X 0,Y 753.38,Z 814.809,A -85,B 0,C 180,E1 35154.197,E2 35154.197} C_VEL
LIN {X 0,Y 753.596,Z 589.172,A -85,B 0,C 180,E1 35151.567,E2 35151.567} C_VEL
LIN {X 0,Y 753.824,Z 375.056,A -85,B 0,C 180,E1 35148.983,E2 35148.983} C_VEL
LIN {X 0,Y 753.672,Z 351.216,A -85,B 0,C 180,E1 35148.677,E2 35148.677} C_VEL
LIN {X 0,Y 753.379,Z 348.793,A -85,B 0,C 180,E1 35148.58,E2 35148.58} C_VEL
LIN {X 0,Y 753.553,Z 302.894,A -85,B 0,C 180,E1 35145.951,E2 35145.951} C_VEL
LIN {X 0,Y 753.398,Z 289.228,A -85,B 0,C 180,E1 35145.13,E2 35145.13} C_VEL
LIN {X 0,Y 752.007,Z 285.776,A -85,B 0,C 180,E1 35144.775,E2 35144.775} C_VEL
LIN {X 0,Y 751.94,Z 285.553,A -85,B 0,C 180,E1 35142.082,E2 35142.082} C_VEL
LIN {X 0,Y 751.966,Z 285.562,A -85,B 0,C 180,E1 35139.267,E2 35139.267} C_VEL
LIN {X 0,Y 751.964,Z 285.553,A -85,B 0,C 180,E1 35136.374,E2 35136.374} C_VEL
LIN {X 0,Y 751.974,Z 285.566,A -85,B 0,C 180,E1 35133.383,E2 35133.383} C_VEL
LIN {X 0,Y 751.976,Z 285.552,A -85,B 0,C 180,E1 35130.35,E2 35130.35} C_VEL
LIN {X 0,Y 751.965,Z 285.564,A -85,B 0,C 180,E1 35127.351,E2 35127.351} C_VEL
LIN {X 0,Y 751.963,Z 285.555,A -85,B 0,C 180,E1 35124.381,E2 35124.381} C_VEL
LIN {X 0,Y 751.95,Z 285.557,A -85,B 0,C 180,E1 35121.531,E2 35121.531} C_VEL
LIN {X 0,Y 751.958,Z 285.563,A -85,B 0,C 180,E1 35118.771,E2 35118.771} C_VEL
LIN {X 0,Y 751.973,Z 285.549,A -85,B 0,C 180,E1 35115.898,E2 35115.898} C_VEL
LIN {X 0,Y 751.972,Z 285.567,A -85,B 0,C 180,E1 35112.908,E2 35112.908} C_VEL
LIN {X 0,Y 751.962,Z 285.55,A -85,B 0,C 180,E1 35109.954,E2 35109.954} C_VEL
LIN {X 0,Y 751.961,Z 285.562,A -85,B 0,C 180,E1 35107.027,E2 35107.027} C_VEL
LIN {X 0,Y 751.944,Z 285.56,A -85,B 0,C 180,E1 35104.234,E2 35104.234} C_VEL
LIN {X 0,Y 751.972,Z 285.553,A -85,B 0,C 180,E1 35101.448,E2 35101.448} C_VEL
LIN {X 0,Y 751.964,Z 285.564,A -85,B 0,C 180,E1 35098.476,E2 35098.476} C_VEL
LIN {X 0,Y 751.965,Z 285.554,A -85,B 0,C 180,E1 35095.5,E2 35095.5} C_VEL
LIN {X 0,Y 751.966,Z 285.565,A -85,B 0,C 180,E1 35094.418,E2 35094.418} C_VEL
LIN {X 0,Y 750.937,Z 285.684,A -85,B 0,C 180,E1 35093.831,E2 35093.831} C_VEL
LIN {X 0,Y 744.52,Z 286.491,A -85,B 0,C 180,E1 35092.188,E2 35092.188} C_VEL
LIN {X 0,Y 744,Z 286.547,A -85,B 0,C 180,E1 35091.761,E2 35091.761} C_VEL
LIN {X 0,Y 744.026,Z 286.546,A -85,B 0,C 180,E1 35088.92,E2 35088.92} C_VEL
LIN {X 0,Y 744.01,Z 286.553,A -85,B 0,C 180,E1 35086.08,E2 35086.08} C_VEL
LIN {X 0,Y 744.019,Z 286.542,A -85,B 0,C 180,E1 35083.205,E2 35083.205} C_VEL
LIN {X 0,Y 744.026,Z 286.554,A -85,B 0,C 180,E1 35080.123,E2 35080.123} C_VEL
LIN {X 0,Y 743.997,Z 286.546,A -85,B 0,C 180,E1 35077.312,E2 35077.312} C_VEL
LIN {X 0,Y 744.029,Z 286.543,A -85,B 0,C 180,E1 35074.444,E2 35074.444} C_VEL
LIN {X 0,Y 743.993,Z 286.551,A -85,B 0,C 180,E1 35071.591,E2 35071.591} C_VEL
LIN {X 0,Y 744.012,Z 286.54,A -85,B 0,C 180,E1 35068.841,E2 35068.841} C_VEL
LIN {X 0,Y 744.012,Z 286.554,A -85,B 0,C 180,E1 35065.729,E2 35065.729} C_VEL
LIN {X 0,Y 743.983,Z 286.543,A -85,B 0,C 180,E1 35063.076,E2 35063.076} C_VEL
LIN {X 0,Y 744.036,Z 286.546,A -85,B 0,C 180,E1 35060.332,E2 35060.332} C_VEL
LIN {X 0,Y 743.997,Z 286.552,A -85,B 0,C 180,E1 35057.43,E2 35057.43} C_VEL
LIN {X 0,Y 743.982,Z 286.548,A -85,B 0,C 180,E1 35054.766,E2 35054.766} C_VEL
LIN {X 0,Y 744.037,Z 286.547,A -85,B 0,C 180,E1 35051.998,E2 35051.998} C_VEL
LIN {X 0,Y 743.985,Z 286.553,A -85,B 0,C 180,E1 35049.152,E2 35049.152} C_VEL
LIN {X 0,Y 743.979,Z 286.547,A -85,B 0,C 180,E1 35046.538,E2 35046.538} C_VEL
LIN {X 0,Y 744.035,Z 286.542,A -85,B 0,C 180,E1 35043.709,E2 35043.709} C_VEL
LIN {X 0,Y 744.003,Z 286.774,A -85,B 0,C 180,E1 35042.579,E2 35042.579} C_VEL
LIN {X 0,Y 746.518,Z 293.344,A -85,B 0,C 180,E1 35041.941,E2 35041.941} C_VEL
LIN {X 0,Y 746.2,Z 334.724,A -85,B 0,C 180,E1 35039.27,E2 35039.27} C_VEL
LIN {X 0,Y 746.232,Z 347.208,A -85,B 0,C 180,E1 35038.5,E2 35038.5} C_VEL
LIN {X 0,Y 747.099,Z 351.652,A -85,B 0,C 180,E1 35038.392,E2 35038.392} C_VEL
LIN {X 0,Y 746.65,Z 592.937,A -85,B 0,C 180,E1 35035.606,E2 35035.606} C_VEL
LIN {X 0,Y 746.324,Z 779.348,A -85,B 0,C 180,E1 35033.491,E2 35033.491} C_VEL
LIN {X 0,Y 746.239,Z 800.898,A -85,B 0,C 180,E1 35033.149,E2 35033.149} C_VEL
LIN {X 0,Y 746.049,Z 828.086,A -85,B 0,C 180,E1 35032.562,E2 35032.562} C_VEL
LIN {X 0,Y 745.913,Z 849.138,A -85,B 0,C 180,E1 35031.982,E2 35031.982} C_VEL
LIN {X 0,Y 745.769,Z 868.723,A -85,B 0,C 180,E1 35031.346,E2 35031.346} C_VEL
LIN {X 0,Y 745.599,Z 892.505,A -85,B 0,C 180,E1 35030.446,E2 35030.446} C_VEL
LIN {X 0,Y 745.343,Z 915.978,A -85,B 0,C 180,E1 35029.391,E2 35029.391} C_VEL
LIN {X 0,Y 745.168,Z 935.728,A -85,B 0,C 180,E1 35028.38,E2 35028.38} C_VEL
LIN {X 0,Y 744.939,Z 958.596,A -85,B 0,C 180,E1 35027.054,E2 35027.054} C_VEL
LIN {X 0,Y 744.762,Z 977.897,A -85,B 0,C 180,E1 35025.775,E2 35025.775} C_VEL
LIN {X 0,Y 744.62,Z 997.309,A -85,B 0,C 180,E1 35024.344,E2 35024.344} C_VEL
LIN {X 0,Y 744.421,Z 1015.721,A -85,B 0,C 180,E1 35022.799,E2 35022.799} C_VEL
LIN {X 0,Y 744.306,Z 1032.487,A -85,B 0,C 180,E1 35021.232,E2 35021.232} C_VEL
LIN {X 0,Y 744.187,Z 1048.66,A -85,B 0,C 180,E1 35019.512,E2 35019.512} C_VEL
LIN {X 0,Y 744.098,Z 1061.066,A -85,B 0,C 180,E1 35018.033,E2 35018.033} C_VEL
LIN {X 0,Y 744.055,Z 1074.403,A -85,B 0,C 180,E1 35016.249,E2 35016.249} C_VEL
LIN {X 0,Y 743.982,Z 1086.243,A -85,B 0,C 180,E1 35014.393,E2 35014.393} C_VEL
LIN {X 0,Y 743.946,Z 1094.821,A -85,B 0,C 180,E1 35012.85,E2 35012.85} C_VEL
LIN {X 0,Y 743.938,Z 1102.605,A -85,B 0,C 180,E1 35011.232,E2 35011.232} C_VEL
LIN {X 0,Y 743.913,Z 1110.838,A -85,B 0,C 180,E1 35009.153,E2 35009.153} C_VEL
LIN {X 0,Y 743.918,Z 1116.065,A -85,B 0,C 180,E1 35007.458,E2 35007.458} C_VEL
LIN {X 0,Y 743.913,Z 1119.993,A -85,B 0,C 180,E1 35005.808,E2 35005.808} C_VEL
LIN {X 0,Y 743.9,Z 1122.932,A -85,B 0,C 180,E1 35004.06,E2 35004.06} C_VEL
LIN {X 0,Y 743.915,Z 1124.714,A -85,B 0,C 180,E1 35001.965,E2 35001.965} C_VEL
LIN {X 0,Y 743.891,Z 1124.825,A -85,B 0,C 180,E1 35000.328,E2 35000.328} C_VEL
LIN {X 0,Y 743.912,Z 1123.838,A -85,B 0,C 180,E1 34998.683,E2 34998.683} C_VEL
LIN {X 0,Y 743.913,Z 1121.2,A -85,B 0,C 180,E1 34996.688,E2 34996.688} C_VEL
LIN {X 0,Y 743.902,Z 1117.008,A -85,B 0,C 180,E1 34994.806,E2 34994.806} C_VEL
LIN {X 0,Y 743.921,Z 1112.303,A -85,B 0,C 180,E1 34993.204,E2 34993.204} C_VEL
LIN {X 0,Y 743.933,Z 1106.43,A -85,B 0,C 180,E1 34991.588,E2 34991.588} C_VEL
LIN {X 0,Y 743.943,Z 1097.781,A -85,B 0,C 180,E1 34989.629,E2 34989.629} C_VEL
LIN {X 0,Y 743.973,Z 1087.974,A -85,B 0,C 180,E1 34987.812,E2 34987.812} C_VEL
LIN {X 0,Y 744.02,Z 1078.673,A -85,B 0,C 180,E1 34986.308,E2 34986.308} C_VEL
LIN {X 0,Y 744.08,Z 1066.837,A -85,B 0,C 180,E1 34984.618,E2 34984.618} C_VEL
LIN {X 0,Y 744.166,Z 1052.263,A -85,B 0,C 180,E1 34982.81,E2 34982.81} C_VEL
LIN {X 0,Y 744.259,Z 1038.689,A -85,B 0,C 180,E1 34981.317,E2 34981.317} C_VEL
LIN {X 0,Y 744.395,Z 1021.967,A -85,B 0,C 180,E1 34979.666,E2 34979.666} C_VEL
LIN {X 0,Y 744.516,Z 1004.395,A -85,B 0,C 180,E1 34978.144,E2 34978.144} C_VEL
LIN {X 0,Y 744.706,Z 985.78,A -85,B 0,C 180,E1 34976.692,E2 34976.692} C_VEL
LIN {X 0,Y 744.888,Z 964.862,A -85,B 0,C 180,E1 34975.259,E2 34975.259} C_VEL
LIN {X 0,Y 745.046,Z 945.839,A -85,B 0,C 180,E1 34974.094,E2 34974.094} C_VEL
LIN {X 0,Y 745.309,Z 921.785,A -85,B 0,C 180,E1 34972.802,E2 34972.802} C_VEL
LIN {X 0,Y 745.482,Z 901.559,A -85,B 0,C 180,E1 34971.856,E2 34971.856} C_VEL
LIN {X 0,Y 745.654,Z 880.289,A -85,B 0,C 180,E1 34970.982,E2 34970.982} C_VEL
LIN {X 0,Y 745.894,Z 854.881,A -85,B 0,C 180,E1 34970.102,E2 34970.102} C_VEL
LIN {X 0,Y 746.038,Z 833.292,A -85,B 0,C 180,E1 34969.484,E2 34969.484} C_VEL
LIN {X 0,Y 746.153,Z 813.096,A -85,B 0,C 180,E1 34969.005,E2 34969.005} C_VEL
LIN {X 0,Y 746.255,Z 791.141,A -85,B 0,C 180,E1 34968.591,E2 34968.591} C_VEL
LIN {X 0,Y 746.373,Z 758.883,A -85,B 0,C 180,E1 34968.17,E2 34968.17} C_VEL
LIN {X 0,Y 746.79,Z 515.609,A -85,B 0,C 180,E1 34965.421,E2 34965.421} C_VEL
LIN {X 0,Y 746.944,Z 350.101,A -85,B 0,C 180,E1 34963.49,E2 34963.49} C_VEL
LIN {X 0,Y 746.149,Z 346.43,A -85,B 0,C 180,E1 34963.376,E2 34963.376} C_VEL
LIN {X 0,Y 746.437,Z 304.043,A -85,B 0,C 180,E1 34960.67,E2 34960.67} C_VEL
LIN {X 0,Y 746.375,Z 292.733,A -85,B 0,C 180,E1 34959.919,E2 34959.919} C_VEL
LIN {X 0,Y 744.06,Z 286.842,A -85,B 0,C 180,E1 34959.349,E2 34959.349} C_VEL
LIN {X 0,Y 744.023,Z 286.532,A -85,B 0,C 180,E1 34958.577,E2 34958.577} C_VEL
LIN {X 0,Y 744.033,Z 286.544,A -85,B 0,C 180,E1 34955.584,E2 34955.584} C_VEL
LIN {X 0,Y 744.007,Z 286.552,A -85,B 0,C 180,E1 34952.701,E2 34952.701} C_VEL
LIN {X 0,Y 744.018,Z 286.548,A -85,B 0,C 180,E1 34949.907,E2 34949.907} C_VEL
LIN {X 0,Y 744.018,Z 286.545,A -85,B 0,C 180,E1 34947.016,E2 34947.016} C_VEL
LIN {X 0,Y 744.033,Z 286.554,A -85,B 0,C 180,E1 34944.113,E2 34944.113} C_VEL
LIN {X 0,Y 744.035,Z 286.539,A -85,B 0,C 180,E1 34941.028,E2 34941.028} C_VEL
LIN {X 0,Y 744.034,Z 286.553,A -85,B 0,C 180,E1 34938.005,E2 34938.005} C_VEL
LIN {X 0,Y 744.034,Z 286.542,A -85,B 0,C 180,E1 34934.935,E2 34934.935} C_VEL
LIN {X 0,Y 744.026,Z 286.55,A -85,B 0,C 180,E1 34931.944,E2 34931.944} C_VEL
LIN {X 0,Y 744.022,Z 286.544,A -85,B 0,C 180,E1 34928.983,E2 34928.983} C_VEL
LIN {X 0,Y 744.011,Z 286.543,A -85,B 0,C 180,E1 34926.172,E2 34926.172} C_VEL
LIN {X 0,Y 744.024,Z 286.551,A -85,B 0,C 180,E1 34923.39,E2 34923.39} C_VEL
LIN {X 0,Y 744.036,Z 286.539,A -85,B 0,C 180,E1 34920.462,E2 34920.462} C_VEL
LIN {X 0,Y 744.033,Z 286.553,A -85,B 0,C 180,E1 34917.458,E2 34917.458} C_VEL
LIN {X 0,Y 744.031,Z 286.542,A -85,B 0,C 180,E1 34914.447,E2 34914.447} C_VEL
LIN {X 0,Y 744.03,Z 286.553,A -85,B 0,C 180,E1 34911.421,E2 34911.421} C_VEL
LIN {X 0,Y 744.013,Z 286.546,A -85,B 0,C 180,E1 34908.527,E2 34908.527} C_VEL
LIN {X 0,Y 744.018,Z 286.544,A -85,B 0,C 180,E1 34905.763,E2 34905.763} C_VEL
LIN {X 0,Y 744.02,Z 286.553,A -85,B 0,C 180,E1 34902.883,E2 34902.883} C_VEL
LIN {X 0,Y 744.036,Z 286.537,A -85,B 0,C 180,E1 34899.941,E2 34899.941} C_VEL
LIN {X 0,Y 744.034,Z 286.551,A -85,B 0,C 180,E1 34896.895,E2 34896.895} C_VEL
LIN {X 0,Y 744.029,Z 286.543,A -85,B 0,C 180,E1 34893.856,E2 34893.856} C_VEL
LIN {X 0,Y 744.031,Z 286.551,A -85,B 0,C 180,E1 34890.802,E2 34890.802} C_VEL
LIN {X 0,Y 744.011,Z 286.546,A -85,B 0,C 180,E1 34887.937,E2 34887.937} C_VEL
LIN {X 0,Y 744.02,Z 286.55,A -85,B 0,C 180,E1 34885.06,E2 34885.06} C_VEL
LIN {X 0,Y 744.007,Z 286.552,A -85,B 0,C 180,E1 34882.205,E2 34882.205} C_VEL
LIN {X 0,Y 744.032,Z 286.546,A -85,B 0,C 180,E1 34879.324,E2 34879.324} C_VEL
LIN {X 0,Y 744.017,Z 286.495,A -85,B 0,C 180,E1 34876.303,E2 34876.303} C_VEL
LIN {X 0,Y 744.037,Z 286.775,A -85,B 0,C 180,E1 34875.775,E2 34875.775} C_VEL
LIN {X 0,Y 745.526,Z 290.297,A -85,B 0,C 180,E1 34875.41,E2 34875.41} C_VEL
LIN {X 0,Y 747.282,Z 293.993,A -85,B 0,C 180,E1 34875.05,E2 34875.05} C_VEL
LIN {X 0,Y 746.96,Z 336.081,A -85,B 0,C 180,E1 34872.588,E2 34872.588} C_VEL
LIN {X 0,Y 747.04,Z 350.595,A -85,B 0,C 180,E1 34871.781,E2 34871.781} C_VEL
LIN {X 0,Y 747.815,Z 355.044,A -85,B 0,C 180,E1 34871.67,E2 34871.67} C_VEL
LIN {X 0,Y 747.369,Z 567.125,A -85,B 0,C 180,E1 34869.079,E2 34869.079} C_VEL
LIN {X 0,Y 746.931,Z 793.249,A -85,B 0,C 180,E1 34866.413,E2 34866.413} C_VEL
LIN {X 0,Y 746.816,Z 832.871,A -85,B 0,C 180,E1 34865.92,E2 34865.92} C_VEL
LIN {X 0,Y 746.66,Z 859.361,A -85,B 0,C 180,E1 34865.439,E2 34865.439} C_VEL
LIN {X 0,Y 746.491,Z 885.517,A -85,B 0,C 180,E1 34864.812,E2 34864.812} C_VEL
LIN {X 0,Y 746.291,Z 912.984,A -85,B 0,C 180,E1 34863.986,E2 34863.986} C_VEL
LIN {X 0,Y 746.014,Z 938.366,A -85,B 0,C 180,E1 34863.058,E2 34863.058} C_VEL
LIN {X 0,Y 745.813,Z 959.697,A -85,B 0,C 180,E1 34862.156,E2 34862.156} C_VEL
LIN {X 0,Y 745.617,Z 979.508,A -85,B 0,C 180,E1 34861.213,E2 34861.213} C_VEL
LIN {X 0,Y 745.411,Z 1001.048,A -85,B 0,C 180,E1 34860.066,E2 34860.066} C_VEL
LIN {X 0,Y 745.12,Z 1024.92,A -85,B 0,C 180,E1 34858.623,E2 34858.623} C_VEL
LIN {X 0,Y 744.926,Z 1043.445,A -85,B 0,C 180,E1 34857.369,E2 34857.369} C_VEL
LIN {X 0,Y 744.78,Z 1061.272,A -85,B 0,C 180,E1 34856.04,E2 34856.04} C_VEL
LIN {X 0,Y 744.531,Z 1083.001,A -85,B 0,C 180,E1 34854.232,E2 34854.232} C_VEL
LIN {X 0,Y 744.424,Z 1098.83,A -85,B 0,C 180,E1 34852.757,E2 34852.757} C_VEL
LIN {X 0,Y 744.287,Z 1114.957,A -85,B 0,C 180,E1 34851.102,E2 34851.102} C_VEL
LIN {X 0,Y 744.155,Z 1131.866,A -85,B 0,C 180,E1 34849.138,E2 34849.138} C_VEL
LIN {X 0,Y 744.097,Z 1144.251,A -85,B 0,C 180,E1 34847.517,E2 34847.517} C_VEL
LIN {X 0,Y 744.02,Z 1154.737,A -85,B 0,C 180,E1 34845.991,E2 34845.991} C_VEL
LIN {X 0,Y 743.999,Z 1164.524,A -85,B 0,C 180,E1 34844.396,E2 34844.396} C_VEL
LIN {X 0,Y 743.961,Z 1174.755,A -85,B 0,C 180,E1 34842.496,E2 34842.496} C_VEL
LIN {X 0,Y 743.933,Z 1184.912,A -85,B 0,C 180,E1 34840.219,E2 34840.219} C_VEL
LIN {X 0,Y 743.923,Z 1191.892,A -85,B 0,C 180,E1 34838.269,E2 34838.269} C_VEL
LIN {X 0,Y 743.916,Z 1197.734,A -85,B 0,C 180,E1 34836.173,E2 34836.173} C_VEL
LIN {X 0,Y 743.909,Z 1201.928,A -85,B 0,C 180,E1 34834.008,E2 34834.008} C_VEL
LIN {X 0,Y 743.912,Z 1204.213,A -85,B 0,C 180,E1 34832.003,E2 34832.003} C_VEL
LIN {X 0,Y 743.898,Z 1204.939,A -85,B 0,C 180,E1 34829.769,E2 34829.769} C_VEL
LIN {X 0,Y 743.908,Z 1203.979,A -85,B 0,C 180,E1 34827.689,E2 34827.689} C_VEL
LIN {X 0,Y 743.912,Z 1201.304,A -85,B 0,C 180,E1 34825.606,E2 34825.606} C_VEL
LIN {X 0,Y 743.919,Z 1197.153,A -85,B 0,C 180,E1 34823.595,E2 34823.595} C_VEL
LIN {X 0,Y 743.924,Z 1191.155,A -85,B 0,C 180,E1 34821.498,E2 34821.498} C_VEL
LIN {X 0,Y 743.919,Z 1183.319,A -85,B 0,C 180,E1 34819.389,E2 34819.389} C_VEL
LIN {X 0,Y 743.966,Z 1173.524,A -85,B 0,C 180,E1 34817.267,E2 34817.267} C_VEL
LIN {X 0,Y 743.999,Z 1164.525,A -85,B 0,C 180,E1 34815.604,E2 34815.604} C_VEL
LIN {X 0,Y 744.02,Z 1154.738,A -85,B 0,C 180,E1 34814.009,E2 34814.009} C_VEL
LIN {X 0,Y 744.097,Z 1144.252,A -85,B 0,C 180,E1 34812.483,E2 34812.483} C_VEL
LIN {X 0,Y 744.155,Z 1131.867,A -85,B 0,C 180,E1 34810.862,E2 34810.862} C_VEL
LIN {X 0,Y 744.287,Z 1114.958,A -85,B 0,C 180,E1 34808.898,E2 34808.898} C_VEL
LIN {X 0,Y 744.423,Z 1098.831,A -85,B 0,C 180,E1 34807.243,E2 34807.243} C_VEL
LIN {X 0,Y 744.541,Z 1082.148,A -85,B 0,C 180,E1 34805.691,E2 34805.691} C_VEL
LIN {X 0,Y 744.781,Z 1061.274,A -85,B 0,C 180,E1 34803.96,E2 34803.96} C_VEL
LIN {X 0,Y 744.926,Z 1043.446,A -85,B 0,C 180,E1 34802.632,E2 34802.632} C_VEL
LIN {X 0,Y 745.123,Z 1024.605,A -85,B 0,C 180,E1 34801.356,E2 34801.356} C_VEL
LIN {X 0,Y 745.415,Z 1000.247,A -85,B 0,C 180,E1 34799.89,E2 34799.89} C_VEL
LIN {X 0,Y 745.618,Z 979.509,A -85,B 0,C 180,E1 34798.787,E2 34798.787} C_VEL
LIN {X 0,Y 745.813,Z 959.701,A -85,B 0,C 180,E1 34797.844,E2 34797.844} C_VEL
LIN {X 0,Y 746.014,Z 938.37,A -85,B 0,C 180,E1 34796.942,E2 34796.942} C_VEL
LIN {X 0,Y 746.299,Z 911.449,A -85,B 0,C 180,E1 34795.966,E2 34795.966} C_VEL
LIN {X 0,Y 746.495,Z 885.166,A -85,B 0,C 180,E1 34795.178,E2 34795.178} C_VEL
LIN {X 0,Y 746.663,Z 858.73,A -85,B 0,C 180,E1 34794.548,E2 34794.548} C_VEL
LIN {X 0,Y 746.817,Z 832.286,A -85,B 0,C 180,E1 34794.071,E2 34794.071} C_VEL
LIN {X 0,Y 746.938,Z 790.17,A -85,B 0,C 180,E1 34793.552,E2 34793.552} C_VEL
LIN {X 0,Y 747.38,Z 562.743,A -85,B 0,C 180,E1 34790.868,E2 34790.868} C_VEL
LIN {X 0,Y 747.815,Z 353.932,A -85,B 0,C 180,E1 34788.316,E2 34788.316} C_VEL
LIN {X 0,Y 746.886,Z 349.201,A -85,B 0,C 180,E1 34788.161,E2 34788.161} C_VEL
LIN {X 0,Y 747.228,Z 303.704,A -85,B 0,C 180,E1 34785.528,E2 34785.528} C_VEL
LIN {X 0,Y 747.224,Z 293.898,A -85,B 0,C 180,E1 34784.94,E2 34784.94} C_VEL
LIN {X 0,Y 745.333,Z 290.011,A -85,B 0,C 180,E1 34784.558,E2 34784.558} C_VEL
LIN {X 0,Y 744.034,Z 286.757,A -85,B 0,C 180,E1 34784.212,E2 34784.212} C_VEL
LIN {X 0,Y 744.023,Z 286.543,A -85,B 0,C 180,E1 34781.653,E2 34781.653} C_VEL
LIN {X 0,Y 744.033,Z 286.542,A -85,B 0,C 180,E1 34778.669,E2 34778.669} C_VEL
LIN {X 0,Y 744.009,Z 286.55,A -85,B 0,C 180,E1 34775.775,E2 34775.775} C_VEL
LIN {X 0,Y 744.019,Z 286.549,A -85,B 0,C 180,E1 34772.976,E2 34772.976} C_VEL
LIN {X 0,Y 744.017,Z 286.544,A -85,B 0,C 180,E1 34770.085,E2 34770.085} C_VEL
LIN {X 0,Y 744.035,Z 286.549,A -85,B 0,C 180,E1 34767.175,E2 34767.175} C_VEL
LIN {X 0,Y 744.034,Z 286.542,A -85,B 0,C 180,E1 34764.113,E2 34764.113} C_VEL
LIN {X 0,Y 744.037,Z 286.548,A -85,B 0,C 180,E1 34761.11,E2 34761.11} C_VEL
LIN {X 0,Y 744.031,Z 286.542,A -85,B 0,C 180,E1 34758.086,E2 34758.086} C_VEL
LIN {X 0,Y 744.027,Z 286.546,A -85,B 0,C 180,E1 34755.113,E2 34755.113} C_VEL
LIN {X 0,Y 744.011,Z 286.546,A -85,B 0,C 180,E1 34752.26,E2 34752.26} C_VEL
LIN {X 0,Y 744.018,Z 286.54,A -85,B 0,C 180,E1 34749.437,E2 34749.437} C_VEL
LIN {X 0,Y 744.019,Z 286.553,A -85,B 0,C 180,E1 34746.559,E2 34746.559} C_VEL
LIN {X 0,Y 744.035,Z 286.541,A -85,B 0,C 180,E1 34743.621,E2 34743.621} C_VEL
LIN {X 0,Y 744.028,Z 286.554,A -85,B 0,C 180,E1 34740.539,E2 34740.539} C_VEL
LIN {X 0,Y 744.028,Z 286.541,A -85,B 0,C 180,E1 34737.535,E2 34737.535} C_VEL
LIN {X 0,Y 744.027,Z 286.553,A -85,B 0,C 180,E1 34734.423,E2 34734.423} C_VEL
LIN {X 0,Y 744,Z 286.547,A -85,B 0,C 180,E1 34731.761,E2 34731.761} C_VEL
LIN {X 0,Y 743.031,Z 286.671,A -85,B 0,C 180,E1 34731.168,E2 34731.168} C_VEL
LIN {X 0,Y 736.637,Z 287.465,A -85,B 0,C 180,E1 34729.506,E2 34729.506} C_VEL
LIN {X 0,Y 736.094,Z 287.532,A -85,B 0,C 180,E1 34729.075,E2 34729.075} C_VEL
LIN {X 0,Y 736.072,Z 287.542,A -85,B 0,C 180,E1 34726.087,E2 34726.087} C_VEL
LIN {X 0,Y 736.083,Z 287.531,A -85,B 0,C 180,E1 34723.182,E2 34723.182} C_VEL
LIN {X 0,Y 736.081,Z 287.542,A -85,B 0,C 180,E1 34720.065,E2 34720.065} C_VEL
LIN {X 0,Y 736.063,Z 287.535,A -85,B 0,C 180,E1 34717.222,E2 34717.222} C_VEL
LIN {X 0,Y 736.092,Z 287.532,A -85,B 0,C 180,E1 34714.321,E2 34714.321} C_VEL
LIN {X 0,Y 736.051,Z 287.539,A -85,B 0,C 180,E1 34711.508,E2 34711.508} C_VEL
LIN {X 0,Y 736.085,Z 287.526,A -85,B 0,C 180,E1 34708.741,E2 34708.741} C_VEL
LIN {X 0,Y 736.069,Z 287.542,A -85,B 0,C 180,E1 34705.679,E2 34705.679} C_VEL
LIN {X 0,Y 736.047,Z 287.529,A -85,B 0,C 180,E1 34703.001,E2 34703.001} C_VEL
LIN {X 0,Y 736.096,Z 287.537,A -85,B 0,C 180,E1 34700.223,E2 34700.223} C_VEL
LIN {X 0,Y 736.05,Z 287.54,A -85,B 0,C 180,E1 34697.322,E2 34697.322} C_VEL
LIN {X 0,Y 736.047,Z 287.536,A -85,B 0,C 180,E1 34694.721,E2 34694.721} C_VEL
LIN {X 0,Y 736.097,Z 287.539,A -85,B 0,C 180,E1 34691.831,E2 34691.831} C_VEL
LIN {X 0,Y 736.042,Z 287.542,A -85,B 0,C 180,E1 34689.073,E2 34689.073} C_VEL
LIN {X 0,Y 736.045,Z 287.535,A -85,B 0,C 180,E1 34686.466,E2 34686.466} C_VEL
LIN {X 0,Y 736.098,Z 287.518,A -85,B 0,C 180,E1 34683.562,E2 34683.562} C_VEL
LIN {X 0,Y 736.083,Z 287.787,A -85,B 0,C 180,E1 34683.057,E2 34683.057} C_VEL
LIN {X 0,Y 739.067,Z 294.911,A -85,B 0,C 180,E1 34682.339,E2 34682.339} C_VEL
LIN {X 0,Y 739.829,Z 297.29,A -85,B 0,C 180,E1 34682.127,E2 34682.127} C_VEL
LIN {X 0,Y 739.359,Z 339.213,A -85,B 0,C 180,E1 34679.399,E2 34679.399} C_VEL
LIN {X 0,Y 739.353,Z 347.035,A -85,B 0,C 180,E1 34678.915,E2 34678.915} C_VEL
LIN {X 0,Y 740.732,Z 353.605,A -85,B 0,C 180,E1 34678.747,E2 34678.747} C_VEL
LIN {X 0,Y 740.054,Z 595.819,A -85,B 0,C 180,E1 34675.926,E2 34675.926} C_VEL
LIN {X 0,Y 739.565,Z 779.627,A -85,B 0,C 180,E1 34673.822,E2 34673.822} C_VEL
LIN {X 0,Y 739.43,Z 802.472,A -85,B 0,C 180,E1 34673.454,E2 34673.454} C_VEL
LIN {X 0,Y 739.149,Z 828.924,A -85,B 0,C 180,E1 34672.869,E2 34672.869} C_VEL
LIN {X 0,Y 738.943,Z 849.903,A -85,B 0,C 180,E1 34672.284,E2 34672.284} C_VEL
LIN {X 0,Y 738.715,Z 871.156,A -85,B 0,C 180,E1 34671.581,E2 34671.581} C_VEL
LIN {X 0,Y 738.385,Z 895.903,A -85,B 0,C 180,E1 34670.614,E2 34670.614} C_VEL
LIN {X 0,Y 738.074,Z 917.312,A -85,B 0,C 180,E1 34669.631,E2 34669.631} C_VEL
LIN {X 0,Y 737.81,Z 937.689,A -85,B 0,C 180,E1 34668.57,E2 34668.57} C_VEL
LIN {X 0,Y 737.439,Z 960.855,A -85,B 0,C 180,E1 34667.192,E2 34667.192} C_VEL
LIN {X 0,Y 737.2,Z 978.822,A -85,B 0,C 180,E1 34665.981,E2 34665.981} C_VEL
LIN {X 0,Y 736.975,Z 998.124,A -85,B 0,C 180,E1 34664.536,E2 34664.536} C_VEL
LIN {X 0,Y 736.687,Z 1016.629,A -85,B 0,C 180,E1 34662.959,E2 34662.959} C_VEL
LIN {X 0,Y 736.513,Z 1033.541,A -85,B 0,C 180,E1 34661.352,E2 34661.352} C_VEL
LIN {X 0,Y 736.323,Z 1049.551,A -85,B 0,C 180,E1 34659.615,E2 34659.615} C_VEL
LIN {X 0,Y 736.197,Z 1062.495,A -85,B 0,C 180,E1 34658.041,E2 34658.041} C_VEL
LIN {X 0,Y 736.087,Z 1076.613,A -85,B 0,C 180,E1 34656.082,E2 34656.082} C_VEL
LIN {X 0,Y 736.02,Z 1086.827,A -85,B 0,C 180,E1 34654.441,E2 34654.441} C_VEL
LIN {X 0,Y 735.972,Z 1095.336,A -85,B 0,C 180,E1 34652.881,E2 34652.881} C_VEL
LIN {X 0,Y 735.954,Z 1104.101,A -85,B 0,C 180,E1 34651.012,E2 34651.012} C_VEL
LIN {X 0,Y 735.927,Z 1111.664,A -85,B 0,C 180,E1 34648.988,E2 34648.988} C_VEL
LIN {X 0,Y 735.915,Z 1116.531,A -85,B 0,C 180,E1 34647.352,E2 34647.352} C_VEL
LIN {X 0,Y 735.899,Z 1120.451,A -85,B 0,C 180,E1 34645.636,E2 34645.636} C_VEL
LIN {X 0,Y 735.914,Z 1123.602,A -85,B 0,C 180,E1 34643.525,E2 34643.525} C_VEL
LIN {X 0,Y 735.914,Z 1124.787,A -85,B 0,C 180,E1 34641.72,E2 34641.72} C_VEL
LIN {X 0,Y 735.893,Z 1124.751,A -85,B 0,C 180,E1 34640.064,E2 34640.064} C_VEL
LIN {X 0,Y 735.905,Z 1123.252,A -85,B 0,C 180,E1 34638.038,E2 34638.038} C_VEL
LIN {X 0,Y 735.895,Z 1120.229,A -85,B 0,C 180,E1 34636.165,E2 34636.165} C_VEL
LIN {X 0,Y 735.923,Z 1116.526,A -85,B 0,C 180,E1 34634.556,E2 34634.556} C_VEL
LIN {X 0,Y 735.908,Z 1111.703,A -85,B 0,C 180,E1 34632.934,E2 34632.934} C_VEL
LIN {X 0,Y 735.942,Z 1104.422,A -85,B 0,C 180,E1 34630.97,E2 34630.97} C_VEL
LIN {X 0,Y 735.968,Z 1095.523,A -85,B 0,C 180,E1 34629.065,E2 34629.065} C_VEL
LIN {X 0,Y 736.021,Z 1086.928,A -85,B 0,C 180,E1 34627.487,E2 34627.487} C_VEL
LIN {X 0,Y 736.098,Z 1076.312,A -85,B 0,C 180,E1 34625.782,E2 34625.782} C_VEL
LIN {X 0,Y 736.201,Z 1062.466,A -85,B 0,C 180,E1 34623.865,E2 34623.865} C_VEL
LIN {X 0,Y 736.322,Z 1049.587,A -85,B 0,C 180,E1 34622.3,E2 34622.3} C_VEL
LIN {X 0,Y 736.521,Z 1033.62,A -85,B 0,C 180,E1 34620.565,E2 34620.565} C_VEL
LIN {X 0,Y 736.699,Z 1016.64,A -85,B 0,C 180,E1 34618.953,E2 34618.953} C_VEL
LIN {X 0,Y 736.934,Z 999.66,A -85,B 0,C 180,E1 34617.501,E2 34617.501} C_VEL
LIN {X 0,Y 737.192,Z 979.398,A -85,B 0,C 180,E1 34615.969,E2 34615.969} C_VEL
LIN {X 0,Y 737.45,Z 960.733,A -85,B 0,C 180,E1 34614.71,E2 34614.71} C_VEL
LIN {X 0,Y 737.817,Z 936.956,A -85,B 0,C 180,E1 34613.3,E2 34613.3} C_VEL
LIN {X 0,Y 738.078,Z 916.586,A -85,B 0,C 180,E1 34612.243,E2 34612.243} C_VEL
LIN {X 0,Y 738.455,Z 893.183,A -85,B 0,C 180,E1 34611.179,E2 34611.179} C_VEL
LIN {X 0,Y 738.729,Z 869.394,A -85,B 0,C 180,E1 34610.267,E2 34610.267} C_VEL
LIN {X 0,Y 738.952,Z 848.232,A -85,B 0,C 180,E1 34609.574,E2 34609.574} C_VEL
LIN {X 0,Y 739.255,Z 823.41,A -85,B 0,C 180,E1 34608.901,E2 34608.901} C_VEL
LIN {X 0,Y 739.44,Z 798.479,A -85,B 0,C 180,E1 34608.386,E2 34608.386} C_VEL
LIN {X 0,Y 739.566,Z 778.11,A -85,B 0,C 180,E1 34608.068,E2 34608.068} C_VEL
LIN {X 0,Y 740.254,Z 522.64,A -85,B 0,C 180,E1 34605.141,E2 34605.141} C_VEL
LIN {X 0,Y 740.562,Z 351.964,A -85,B 0,C 180,E1 34603.133,E2 34603.133} C_VEL
LIN {X 0,Y 739.314,Z 346.512,A -85,B 0,C 180,E1 34602.972,E2 34602.972} C_VEL
LIN {X 0,Y 739.75,Z 304.326,A -85,B 0,C 180,E1 34600.248,E2 34600.248} C_VEL
LIN {X 0,Y 739.705,Z 296.562,A -85,B 0,C 180,E1 34599.725,E2 34599.725} C_VEL
LIN {X 0,Y 736.117,Z 287.868,A -85,B 0,C 180,E1 34598.87,E2 34598.87} C_VEL
LIN {X 0,Y 736.094,Z 287.517,A -85,B 0,C 180,E1 34598.373,E2 34598.373} C_VEL
LIN {X 0,Y 736.089,Z 287.533,A -85,B 0,C 180,E1 34595.357,E2 34595.357} C_VEL
LIN {X 0,Y 736.092,Z 287.543,A -85,B 0,C 180,E1 34592.341,E2 34592.341} C_VEL
LIN {X 0,Y 736.098,Z 287.527,A -85,B 0,C 180,E1 34589.276,E2 34589.276} C_VEL
LIN {X 0,Y 736.086,Z 287.539,A -85,B 0,C 180,E1 34586.285,E2 34586.285} C_VEL
LIN {X 0,Y 736.092,Z 287.533,A -85,B 0,C 180,E1 34583.284,E2 34583.284} C_VEL
LIN {X 0,Y 736.071,Z 287.535,A -85,B 0,C 180,E1 34580.401,E2 34580.401} C_VEL
LIN {X 0,Y 736.078,Z 287.532,A -85,B 0,C 180,E1 34577.552,E2 34577.552} C_VEL
LIN {X 0,Y 736.084,Z 287.533,A -85,B 0,C 180,E1 34574.716,E2 34574.716} C_VEL
LIN {X 0,Y 736.096,Z 287.536,A -85,B 0,C 180,E1 34571.757,E2 34571.757} C_VEL
LIN {X 0,Y 736.093,Z 287.531,A -85,B 0,C 180,E1 34568.672,E2 34568.672} C_VEL
LIN {X 0,Y 736.096,Z 287.54,A -85,B 0,C 180,E1 34565.613,E2 34565.613} C_VEL
LIN {X 0,Y 736.095,Z 287.528,A -85,B 0,C 180,E1 34562.569,E2 34562.569} C_VEL
LIN {X 0,Y 736.098,Z 287.541,A -85,B 0,C 180,E1 34559.533,E2 34559.533} C_VEL
LIN {X 0,Y 736.091,Z 287.525,A -85,B 0,C 180,E1 34556.495,E2 34556.495} C_VEL
LIN {X 0,Y 736.093,Z 287.542,A -85,B 0,C 180,E1 34553.448,E2 34553.448} C_VEL
LIN {X 0,Y 736.081,Z 287.527,A -85,B 0,C 180,E1 34550.461,E2 34550.461} C_VEL
LIN {X 0,Y 736.077,Z 287.539,A -85,B 0,C 180,E1 34547.597,E2 34547.597} C_VEL
LIN {X 0,Y 736.073,Z 287.538,A -85,B 0,C 180,E1 34544.801,E2 34544.801} C_VEL
LIN {X 0,Y 736.094,Z 287.531,A -85,B 0,C 180,E1 34541.958,E2 34541.958} C_VEL
LIN {X 0,Y 736.09,Z 287.543,A -85,B 0,C 180,E1 34538.901,E2 34538.901} C_VEL
LIN {X 0,Y 736.095,Z 287.526,A -85,B 0,C 180,E1 34535.866,E2 34535.866} C_VEL
LIN {X 0,Y 736.09,Z 287.54,A -85,B 0,C 180,E1 34532.756,E2 34532.756} C_VEL
LIN {X 0,Y 736.094,Z 287.532,A -85,B 0,C 180,E1 34529.738,E2 34529.738} C_VEL
LIN {X 0,Y 736.091,Z 287.543,A -85,B 0,C 180,E1 34526.623,E2 34526.623} C_VEL
LIN {X 0,Y 736.084,Z 287.535,A -85,B 0,C 180,E1 34523.659,E2 34523.659} C_VEL
LIN {X 0,Y 736.091,Z 287.536,A -85,B 0,C 180,E1 34520.614,E2 34520.614} C_VEL
LIN {X 0,Y 736.064,Z 287.521,A -85,B 0,C 180,E1 34517.745,E2 34517.745} C_VEL
LIN {X 0,Y 736.113,Z 287.695,A -85,B 0,C 180,E1 34516.367,E2 34516.367} C_VEL
LIN {X 0,Y 737.309,Z 290.882,A -85,B 0,C 180,E1 34516.025,E2 34516.025} C_VEL
LIN {X 0,Y 741.003,Z 298.298,A -85,B 0,C 180,E1 34515.275,E2 34515.275} C_VEL
LIN {X 0,Y 740.487,Z 341.555,A -85,B 0,C 180,E1 34512.729,E2 34512.729} C_VEL
LIN {X 0,Y 740.578,Z 350.609,A -85,B 0,C 180,E1 34512.229,E2 34512.229} C_VEL
LIN {X 0,Y 741.82,Z 356.779,A -85,B 0,C 180,E1 34512.062,E2 34512.062} C_VEL
LIN {X 0,Y 741.142,Z 568.803,A -85,B 0,C 180,E1 34509.451,E2 34509.451} C_VEL
LIN {X 0,Y 740.479,Z 794.742,A -85,B 0,C 180,E1 34506.764,E2 34506.764} C_VEL
LIN {X 0,Y 740.311,Z 833.466,A -85,B 0,C 180,E1 34506.277,E2 34506.277} C_VEL
LIN {X 0,Y 740.077,Z 860.041,A -85,B 0,C 180,E1 34505.787,E2 34505.787} C_VEL
LIN {X 0,Y 739.823,Z 885.955,A -85,B 0,C 180,E1 34505.16,E2 34505.16} C_VEL
LIN {X 0,Y 739.516,Z 913.629,A -85,B 0,C 180,E1 34504.319,E2 34504.319} C_VEL
LIN {X 0,Y 739.093,Z 939.488,A -85,B 0,C 180,E1 34503.362,E2 34503.362} C_VEL
LIN {X 0,Y 738.79,Z 960.694,A -85,B 0,C 180,E1 34502.453,E2 34502.453} C_VEL
LIN {X 0,Y 738.489,Z 981.246,A -85,B 0,C 180,E1 34501.46,E2 34501.46} C_VEL
LIN {X 0,Y 738.11,Z 1005.695,A -85,B 0,C 180,E1 34500.125,E2 34500.125} C_VEL
LIN {X 0,Y 737.732,Z 1026.908,A -85,B 0,C 180,E1 34498.804,E2 34498.804} C_VEL
LIN {X 0,Y 737.449,Z 1045.338,A -85,B 0,C 180,E1 34497.533,E2 34497.533} C_VEL
LIN {X 0,Y 737.182,Z 1066.23,A -85,B 0,C 180,E1 34495.937,E2 34495.937} C_VEL
LIN {X 0,Y 736.85,Z 1085.146,A -85,B 0,C 180,E1 34494.305,E2 34494.305} C_VEL
LIN {X 0,Y 736.681,Z 1100.567,A -85,B 0,C 180,E1 34492.838,E2 34492.838} C_VEL
LIN {X 0,Y 736.469,Z 1117.989,A -85,B 0,C 180,E1 34491.003,E2 34491.003} C_VEL
LIN {X 0,Y 736.294,Z 1132.513,A -85,B 0,C 180,E1 34489.268,E2 34489.268} C_VEL
LIN {X 0,Y 736.196,Z 1144.253,A -85,B 0,C 180,E1 34487.711,E2 34487.711} C_VEL
LIN {X 0,Y 736.091,Z 1154.738,A -85,B 0,C 180,E1 34486.168,E2 34486.168} C_VEL
LIN {X 0,Y 736.045,Z 1164.525,A -85,B 0,C 180,E1 34484.555,E2 34484.555} C_VEL
LIN {X 0,Y 735.988,Z 1174.755,A -85,B 0,C 180,E1 34482.634,E2 34482.634} C_VEL
LIN {X 0,Y 735.948,Z 1184.913,A -85,B 0,C 180,E1 34480.331,E2 34480.331} C_VEL
LIN {X 0,Y 735.928,Z 1192.136,A -85,B 0,C 180,E1 34478.28,E2 34478.28} C_VEL
LIN {X 0,Y 735.918,Z 1197.735,A -85,B 0,C 180,E1 34476.24,E2 34476.24} C_VEL
LIN {X 0,Y 735.912,Z 1201.928,A -85,B 0,C 180,E1 34474.051,E2 34474.051} C_VEL
LIN {X 0,Y 735.912,Z 1204.213,A -85,B 0,C 180,E1 34472.024,E2 34472.024} C_VEL
LIN {X 0,Y 735.898,Z 1204.939,A -85,B 0,C 180,E1 34469.767,E2 34469.767} C_VEL
LIN {X 0,Y 735.908,Z 1203.976,A -85,B 0,C 180,E1 34467.664,E2 34467.664} C_VEL
LIN {X 0,Y 735.91,Z 1201.303,A -85,B 0,C 180,E1 34465.558,E2 34465.558} C_VEL
LIN {X 0,Y 735.92,Z 1197.153,A -85,B 0,C 180,E1 34463.525,E2 34463.525} C_VEL
LIN {X 0,Y 735.931,Z 1191.151,A -85,B 0,C 180,E1 34461.405,E2 34461.405} C_VEL
LIN {X 0,Y 735.931,Z 1183.319,A -85,B 0,C 180,E1 34459.273,E2 34459.273} C_VEL
LIN {X 0,Y 735.999,Z 1173.526,A -85,B 0,C 180,E1 34457.127,E2 34457.127} C_VEL
LIN {X 0,Y 736.045,Z 1164.527,A -85,B 0,C 180,E1 34455.445,E2 34455.445} C_VEL
LIN {X 0,Y 736.092,Z 1154.646,A -85,B 0,C 180,E1 34453.817,E2 34453.817} C_VEL
LIN {X 0,Y 736.198,Z 1143.672,A -85,B 0,C 180,E1 34452.207,E2 34452.207} C_VEL
LIN {X 0,Y 736.364,Z 1129.29,A -85,B 0,C 180,E1 34450.322,E2 34450.322} C_VEL
LIN {X 0,Y 736.522,Z 1112.62,A -85,B 0,C 180,E1 34448.414,E2 34448.414} C_VEL
LIN {X 0,Y 736.685,Z 1097.979,A -85,B 0,C 180,E1 34446.906,E2 34446.906} C_VEL
LIN {X 0,Y 736.985,Z 1079.52,A -85,B 0,C 180,E1 34445.184,E2 34445.184} C_VEL
LIN {X 0,Y 737.229,Z 1060.167,A -85,B 0,C 180,E1 34443.587,E2 34443.587} C_VEL
LIN {X 0,Y 737.478,Z 1042.501,A -85,B 0,C 180,E1 34442.263,E2 34442.263} C_VEL
LIN {X 0,Y 737.895,Z 1020.413,A -85,B 0,C 180,E1 34440.77,E2 34440.77} C_VEL
LIN {X 0,Y 738.221,Z 997.841,A -85,B 0,C 180,E1 34439.431,E2 34439.431} C_VEL
LIN {X 0,Y 738.518,Z 977.732,A -85,B 0,C 180,E1 34438.362,E2 34438.362} C_VEL
LIN {X 0,Y 738.84,Z 956.624,A -85,B 0,C 180,E1 34437.361,E2 34437.361} C_VEL
LIN {X 0,Y 739.293,Z 929.68,A -85,B 0,C 180,E1 34436.257,E2 34436.257} C_VEL
LIN {X 0,Y 739.567,Z 907.053,A -85,B 0,C 180,E1 34435.472,E2 34435.472} C_VEL
LIN {X 0,Y 739.849,Z 883.683,A -85,B 0,C 180,E1 34434.78,E2 34434.78} C_VEL
LIN {X 0,Y 740.115,Z 856.873,A -85,B 0,C 180,E1 34434.145,E2 34434.145} C_VEL
LIN {X 0,Y 740.323,Z 829.71,A -85,B 0,C 180,E1 34433.667,E2 34433.667} C_VEL
LIN {X 0,Y 740.657,Z 731.551,A -85,B 0,C 180,E1 34432.493,E2 34432.493} C_VEL
LIN {X 0,Y 741.331,Z 509.394,A -85,B 0,C 180,E1 34429.827,E2 34429.827} C_VEL
LIN {X 0,Y 741.695,Z 355.394,A -85,B 0,C 180,E1 34427.912,E2 34427.912} C_VEL
LIN {X 0,Y 740.434,Z 349.617,A -85,B 0,C 180,E1 34427.734,E2 34427.734} C_VEL
LIN {X 0,Y 740.938,Z 304.694,A -85,B 0,C 180,E1 34425.109,E2 34425.109} C_VEL
LIN {X 0,Y 740.817,Z 297.878,A -85,B 0,C 180,E1 34424.685,E2 34424.685} C_VEL
LIN {X 0,Y 737.309,Z 290.882,A -85,B 0,C 180,E1 34423.975,E2 34423.975} C_VEL
LIN {X 0,Y 736.118,Z 287.732,A -85,B 0,C 180,E1 34423.633,E2 34423.633} C_VEL
LIN {X 0,Y 736.086,Z 287.54,A -85,B 0,C 180,E1 34420.9,E2 34420.9} C_VEL
LIN {X 0,Y 736.067,Z 287.535,A -85,B 0,C 180,E1 34418.078,E2 34418.078} C_VEL
LIN {X 0,Y 736.095,Z 287.542,A -85,B 0,C 180,E1 34415.262,E2 34415.262} C_VEL
LIN {X 0,Y 736.089,Z 287.53,A -85,B 0,C 180,E1 34412.266,E2 34412.266} C_VEL
LIN {X 0,Y 736.097,Z 287.543,A -85,B 0,C 180,E1 34409.276,E2 34409.276} C_VEL
LIN {X 0,Y 736.093,Z 287.527,A -85,B 0,C 180,E1 34406.198,E2 34406.198} C_VEL
LIN {X 0,Y 736.093,Z 287.54,A -85,B 0,C 180,E1 34403.134,E2 34403.134} C_VEL
LIN {X 0,Y 736.095,Z 287.53,A -85,B 0,C 180,E1 34400.101,E2 34400.101} C_VEL
LIN {X 0,Y 736.095,Z 287.537,A -85,B 0,C 180,E1 34397.009,E2 34397.009} C_VEL
LIN {X 0,Y 736.091,Z 287.53,A -85,B 0,C 180,E1 34393.992,E2 34393.992} C_VEL
LIN {X 0,Y 736.092,Z 287.54,A -85,B 0,C 180,E1 34390.963,E2 34390.963} C_VEL
LIN {X 0,Y 736.076,Z 287.532,A -85,B 0,C 180,E1 34388.01,E2 34388.01} C_VEL
LIN {X 0,Y 736.08,Z 287.538,A -85,B 0,C 180,E1 34385.144,E2 34385.144} C_VEL
LIN {X 0,Y 736.071,Z 287.539,A -85,B 0,C 180,E1 34382.336,E2 34382.336} C_VEL
LIN {X 0,Y 736.098,Z 287.531,A -85,B 0,C 180,E1 34379.455,E2 34379.455} C_VEL
LIN {X 0,Y 736.085,Z 287.543,A -85,B 0,C 180,E1 34376.417,E2 34376.417} C_VEL
LIN {X 0,Y 736.086,Z 287.531,A -85,B 0,C 180,E1 34373.448,E2 34373.448} C_VEL
LIN {X 0,Y 736.092,Z 287.542,A -85,B 0,C 180,E1 34370.382,E2 34370.382} C_VEL
LIN {X 0,Y 736.094,Z 287.532,A -85,B 0,C 180,E1 34369.075,E2 34369.075} C_VEL
LIN {X 0,Y 735.091,Z 287.669,A -85,B 0,C 180,E1 34368.475,E2 34368.475} C_VEL
LIN {X 0,Y 728.686,Z 288.461,A -85,B 0,C 180,E1 34366.796,E2 34366.796} C_VEL
LIN {X 0,Y 728.158,Z 288.53,A -85,B 0,C 180,E1 34366.36,E2 34366.36} C_VEL
LIN {X 0,Y 728.121,Z 288.522,A -85,B 0,C 180,E1 34363.485,E2 34363.485} C_VEL
LIN {X 0,Y 728.15,Z 288.527,A -85,B 0,C 180,E1 34360.622,E2 34360.622} C_VEL
LIN {X 0,Y 728.12,Z 288.529,A -85,B 0,C 180,E1 34357.75,E2 34357.75} C_VEL
LIN {X 0,Y 728.147,Z 288.512,A -85,B 0,C 180,E1 34354.892,E2 34354.892} C_VEL
LIN {X 0,Y 728.131,Z 288.531,A -85,B 0,C 180,E1 34351.81,E2 34351.81} C_VEL
LIN {X 0,Y 728.12,Z 288.516,A -85,B 0,C 180,E1 34349.004,E2 34349.004} C_VEL
LIN {X 0,Y 728.157,Z 288.531,A -85,B 0,C 180,E1 34346.021,E2 34346.021} C_VEL
LIN {X 0,Y 728.105,Z 288.518,A -85,B 0,C 180,E1 34343.219,E2 34343.219} C_VEL
LIN {X 0,Y 728.157,Z 288.524,A -85,B 0,C 180,E1 34340.383,E2 34340.383} C_VEL
LIN {X 0,Y 728.116,Z 288.53,A -85,B 0,C 180,E1 34337.389,E2 34337.389} C_VEL
LIN {X 0,Y 728.111,Z 288.525,A -85,B 0,C 180,E1 34334.675,E2 34334.675} C_VEL
LIN {X 0,Y 728.16,Z 288.529,A -85,B 0,C 180,E1 34331.757,E2 34331.757} C_VEL
LIN {X 0,Y 728.099,Z 288.53,A -85,B 0,C 180,E1 34328.972,E2 34328.972} C_VEL
LIN {X 0,Y 728.113,Z 288.523,A -85,B 0,C 180,E1 34326.386,E2 34326.386} C_VEL
LIN {X 0,Y 728.185,Z 288.692,A -85,B 0,C 180,E1 34323.574,E2 34323.574} C_VEL
LIN {X 0,Y 729.503,Z 292.11,A -85,B 0,C 180,E1 34323.198,E2 34323.198} C_VEL
LIN {X 0,Y 733.152,Z 300.86,A -85,B 0,C 180,E1 34322.342,E2 34322.342} C_VEL
LIN {X 0,Y 732.529,Z 342.654,A -85,B 0,C 180,E1 34319.6,E2 34319.6} C_VEL
LIN {X 0,Y 732.527,Z 346.839,A -85,B 0,C 180,E1 34319.341,E2 34319.341} C_VEL
LIN {X 0,Y 734.393,Z 355.429,A -85,B 0,C 180,E1 34319.109,E2 34319.109} C_VEL
LIN {X 0,Y 733.484,Z 598.235,A -85,B 0,C 180,E1 34316.258,E2 34316.258} C_VEL
LIN {X 0,Y 732.831,Z 779.711,A -85,B 0,C 180,E1 34314.162,E2 34314.162} C_VEL
LIN {X 0,Y 732.646,Z 803.448,A -85,B 0,C 180,E1 34313.775,E2 34313.775} C_VEL
LIN {X 0,Y 732.273,Z 829.435,A -85,B 0,C 180,E1 34313.191,E2 34313.191} C_VEL
LIN {X 0,Y 731.994,Z 850.667,A -85,B 0,C 180,E1 34312.592,E2 34312.592} C_VEL
LIN {X 0,Y 731.675,Z 873.617,A -85,B 0,C 180,E1 34311.82,E2 34311.82} C_VEL
LIN {X 0,Y 731.195,Z 898.319,A -85,B 0,C 180,E1 34310.826,E2 34310.826} C_VEL
LIN {X 0,Y 730.819,Z 918.644,A -85,B 0,C 180,E1 34309.876,E2 34309.876} C_VEL
LIN {X 0,Y 730.442,Z 941.135,A -85,B 0,C 180,E1 34308.681,E2 34308.681} C_VEL
LIN {X 0,Y 729.96,Z 962.487,A -85,B 0,C 180,E1 34307.374,E2 34307.374} C_VEL
LIN {X 0,Y 729.633,Z 981.458,A -85,B 0,C 180,E1 34306.07,E2 34306.07} C_VEL
LIN {X 0,Y 729.263,Z 1001.314,A -85,B 0,C 180,E1 34304.531,E2 34304.531} C_VEL
LIN {X 0,Y 728.955,Z 1017.989,A -85,B 0,C 180,E1 34303.08,E2 34303.08} C_VEL
LIN {X 0,Y 728.674,Z 1036.043,A -85,B 0,C 180,E1 34301.316,E2 34301.316} C_VEL
LIN {X 0,Y 728.463,Z 1050.441,A -85,B 0,C 180,E1 34299.719,E2 34299.719} C_VEL
LIN {X 0,Y 728.295,Z 1063.921,A -85,B 0,C 180,E1 34298.05,E2 34298.05} C_VEL
LIN {X 0,Y 728.15,Z 1077.269,A -85,B 0,C 180,E1 34296.148,E2 34296.148} C_VEL
LIN {X 0,Y 728.059,Z 1086.958,A -85,B 0,C 180,E1 34294.569,E2 34294.569} C_VEL
LIN {X 0,Y 727.997,Z 1095.85,A -85,B 0,C 180,E1 34292.913,E2 34292.913} C_VEL
LIN {X 0,Y 727.957,Z 1104.847,A -85,B 0,C 180,E1 34290.944,E2 34290.944} C_VEL
LIN {X 0,Y 727.93,Z 1111.732,A -85,B 0,C 180,E1 34289.056,E2 34289.056} C_VEL
LIN {X 0,Y 727.919,Z 1116.586,A -85,B 0,C 180,E1 34287.402,E2 34287.402} C_VEL
LIN {X 0,Y 727.901,Z 1120.493,A -85,B 0,C 180,E1 34285.667,E2 34285.667} C_VEL
LIN {X 0,Y 727.914,Z 1123.62,A -85,B 0,C 180,E1 34283.533,E2 34283.533} C_VEL
LIN {X 0,Y 727.914,Z 1124.793,A -85,B 0,C 180,E1 34281.707,E2 34281.707} C_VEL
LIN {X 0,Y 727.898,Z 1124.722,A -85,B 0,C 180,E1 34279.953,E2 34279.953} C_VEL
LIN {X 0,Y 727.911,Z 1122.94,A -85,B 0,C 180,E1 34277.788,E2 34277.788} C_VEL
LIN {X 0,Y 727.897,Z 1120.023,A -85,B 0,C 180,E1 34276.01,E2 34276.01} C_VEL
LIN {X 0,Y 727.915,Z 1116.172,A -85,B 0,C 180,E1 34274.349,E2 34274.349} C_VEL
LIN {X 0,Y 727.934,Z 1110.575,A -85,B 0,C 180,E1 34272.494,E2 34272.494} C_VEL
LIN {X 0,Y 727.973,Z 1102.471,A -85,B 0,C 180,E1 34270.42,E2 34270.42} C_VEL
LIN {X 0,Y 727.991,Z 1094.975,A -85,B 0,C 180,E1 34268.825,E2 34268.825} C_VEL
LIN {X 0,Y 728.077,Z 1086.233,A -85,B 0,C 180,E1 34267.215,E2 34267.215} C_VEL
LIN {X 0,Y 728.203,Z 1074.465,A -85,B 0,C 180,E1 34265.329,E2 34265.329} C_VEL
LIN {X 0,Y 728.326,Z 1061.122,A -85,B 0,C 180,E1 34263.502,E2 34263.502} C_VEL
LIN {X 0,Y 728.506,Z 1048.092,A -85,B 0,C 180,E1 34261.916,E2 34261.916} C_VEL
LIN {X 0,Y 728.762,Z 1030.6,A -85,B 0,C 180,E1 34260.039,E2 34260.039} C_VEL
LIN {X 0,Y 729.015,Z 1014.928,A -85,B 0,C 180,E1 34258.552,E2 34258.552} C_VEL
LIN {X 0,Y 729.365,Z 995.865,A -85,B 0,C 180,E1 34256.934,E2 34256.934} C_VEL
LIN {X 0,Y 729.691,Z 977.177,A -85,B 0,C 180,E1 34255.534,E2 34255.534} C_VEL
LIN {X 0,Y 730.154,Z 956.046,A -85,B 0,C 180,E1 34254.12,E2 34254.12} C_VEL
LIN {X 0,Y 730.515,Z 934.068,A -85,B 0,C 180,E1 34252.839,E2 34252.839} C_VEL
LIN {X 0,Y 730.943,Z 913.058,A -85,B 0,C 180,E1 34251.759,E2 34251.759} C_VEL
LIN {X 0,Y 731.401,Z 888.346,A -85,B 0,C 180,E1 34250.663,E2 34250.663} C_VEL
LIN {X 0,Y 731.738,Z 866.534,A -85,B 0,C 180,E1 34249.838,E2 34249.838} C_VEL
LIN {X 0,Y 732.099,Z 843.964,A -85,B 0,C 180,E1 34249.113,E2 34249.113} C_VEL
LIN {X 0,Y 732.46,Z 818.039,A -85,B 0,C 180,E1 34248.445,E2 34248.445} C_VEL
LIN {X 0,Y 732.674,Z 796.475,A -85,B 0,C 180,E1 34248.011,E2 34248.011} C_VEL
LIN {X 0,Y 732.845,Z 775.745,A -85,B 0,C 180,E1 34247.695,E2 34247.695} C_VEL
LIN {X 0,Y 733.754,Z 524.321,A -85,B 0,C 180,E1 34244.794,E2 34244.794} C_VEL
LIN {X 0,Y 734.231,Z 353.91,A -85,B 0,C 180,E1 34242.773,E2 34242.773} C_VEL
LIN {X 0,Y 732.506,Z 346.538,A -85,B 0,C 180,E1 34242.556,E2 34242.556} C_VEL
LIN {X 0,Y 733.09,Z 304.889,A -85,B 0,C 180,E1 34239.837,E2 34239.837} C_VEL
LIN {X 0,Y 733.026,Z 300.274,A -85,B 0,C 180,E1 34239.519,E2 34239.519} C_VEL
LIN {X 0,Y 728.198,Z 288.809,A -85,B 0,C 180,E1 34238.363,E2 34238.363} C_VEL
LIN {X 0,Y 728.144,Z 288.53,A -85,B 0,C 180,E1 34237.339,E2 34237.339} C_VEL
LIN {X 0,Y 728.155,Z 288.532,A -85,B 0,C 180,E1 34234.359,E2 34234.359} C_VEL
LIN {X 0,Y 728.153,Z 288.524,A -85,B 0,C 180,E1 34231.27,E2 34231.27} C_VEL
LIN {X 0,Y 728.16,Z 288.53,A -85,B 0,C 180,E1 34228.189,E2 34228.189} C_VEL
LIN {X 0,Y 728.152,Z 288.518,A -85,B 0,C 180,E1 34225.107,E2 34225.107} C_VEL
LIN {X 0,Y 728.157,Z 288.524,A -85,B 0,C 180,E1 34222.049,E2 34222.049} C_VEL
LIN {X 0,Y 728.155,Z 288.521,A -85,B 0,C 180,E1 34218.993,E2 34218.993} C_VEL
LIN {X 0,Y 728.155,Z 288.524,A -85,B 0,C 180,E1 34215.94,E2 34215.94} C_VEL
LIN {X 0,Y 728.156,Z 288.516,A -85,B 0,C 180,E1 34212.853,E2 34212.853} C_VEL
LIN {X 0,Y 728.156,Z 288.531,A -85,B 0,C 180,E1 34209.804,E2 34209.804} C_VEL
LIN {X 0,Y 728.155,Z 288.512,A -85,B 0,C 180,E1 34206.703,E2 34206.703} C_VEL
LIN {X 0,Y 728.156,Z 288.532,A -85,B 0,C 180,E1 34203.622,E2 34203.622} C_VEL
LIN {X 0,Y 728.157,Z 288.516,A -85,B 0,C 180,E1 34200.551,E2 34200.551} C_VEL
LIN {X 0,Y 728.155,Z 288.528,A -85,B 0,C 180,E1 34197.481,E2 34197.481} C_VEL
LIN {X 0,Y 728.155,Z 288.519,A -85,B 0,C 180,E1 34194.405,E2 34194.405} C_VEL
LIN {X 0,Y 728.155,Z 288.524,A -85,B 0,C 180,E1 34191.312,E2 34191.312} C_VEL
LIN {X 0,Y 728.154,Z 288.521,A -85,B 0,C 180,E1 34188.251,E2 34188.251} C_VEL
LIN {X 0,Y 728.158,Z 288.522,A -85,B 0,C 180,E1 34185.169,E2 34185.169} C_VEL
LIN {X 0,Y 728.153,Z 288.521,A -85,B 0,C 180,E1 34182.099,E2 34182.099} C_VEL
LIN {X 0,Y 728.154,Z 288.528,A -85,B 0,C 180,E1 34178.998,E2 34178.998} C_VEL
LIN {X 0,Y 728.143,Z 288.515,A -85,B 0,C 180,E1 34176.017,E2 34176.017} C_VEL
LIN {X 0,Y 728.155,Z 288.533,A -85,B 0,C 180,E1 34172.966,E2 34172.966} C_VEL
LIN {X 0,Y 728.133,Z 288.525,A -85,B 0,C 180,E1 34170.052,E2 34170.052} C_VEL
LIN {X 0,Y 728.144,Z 288.528,A -85,B 0,C 180,E1 34167.18,E2 34167.18} C_VEL
LIN {X 0,Y 728.132,Z 288.532,A -85,B 0,C 180,E1 34164.294,E2 34164.294} C_VEL
LIN {X 0,Y 728.157,Z 288.523,A -85,B 0,C 180,E1 34161.381,E2 34161.381} C_VEL
LIN {X 0,Y 728.142,Z 288.513,A -85,B 0,C 180,E1 34158.331,E2 34158.331} C_VEL
LIN {X 0,Y 728.175,Z 288.722,A -85,B 0,C 180,E1 34156.957,E2 34156.957} C_VEL
LIN {X 0,Y 729.559,Z 292.096,A -85,B 0,C 180,E1 34156.582,E2 34156.582} C_VEL
LIN {X 0,Y 734.735,Z 302.603,A -85,B 0,C 180,E1 34155.504,E2 34155.504} C_VEL
LIN {X 0,Y 734.019,Z 347.027,A -85,B 0,C 180,E1 34152.872,E2 34152.872} C_VEL
LIN {X 0,Y 734.209,Z 350.892,A -85,B 0,C 180,E1 34152.676,E2 34152.676} C_VEL
LIN {X 0,Y 735.858,Z 358.769,A -85,B 0,C 180,E1 34152.456,E2 34152.456} C_VEL
LIN {X 0,Y 734.947,Z 570.457,A -85,B 0,C 180,E1 34149.829,E2 34149.829} C_VEL
LIN {X 0,Y 734.056,Z 795.922,A -85,B 0,C 180,E1 34147.125,E2 34147.125} C_VEL
LIN {X 0,Y 733.835,Z 834.178,A -85,B 0,C 180,E1 34146.638,E2 34146.638} C_VEL
LIN {X 0,Y 733.517,Z 861.131,A -85,B 0,C 180,E1 34146.134,E2 34146.134} C_VEL
LIN {X 0,Y 733.174,Z 886.972,A -85,B 0,C 180,E1 34145.498,E2 34145.498} C_VEL
LIN {X 0,Y 732.728,Z 915.13,A -85,B 0,C 180,E1 34144.627,E2 34144.627} C_VEL
LIN {X 0,Y 732.218,Z 939.49,A -85,B 0,C 180,E1 34143.717,E2 34143.717} C_VEL
LIN {X 0,Y 731.801,Z 960.598,A -85,B 0,C 180,E1 34142.807,E2 34142.807} C_VEL
LIN {X 0,Y 731.387,Z 982.095,A -85,B 0,C 180,E1 34141.757,E2 34141.757} C_VEL
LIN {X 0,Y 730.853,Z 1007.162,A -85,B 0,C 180,E1 34140.365,E2 34140.365} C_VEL
LIN {X 0,Y 730.377,Z 1027.573,A -85,B 0,C 180,E1 34139.077,E2 34139.077} C_VEL
LIN {X 0,Y 729.986,Z 1046.471,A -85,B 0,C 180,E1 34137.755,E2 34137.755} C_VEL
LIN {X 0,Y 729.555,Z 1068.743,A -85,B 0,C 180,E1 34136.012,E2 34136.012} C_VEL
LIN {X 0,Y 729.183,Z 1085.986,A -85,B 0,C 180,E1 34134.5,E2 34134.5} C_VEL
LIN {X 0,Y 728.939,Z 1102.247,A -85,B 0,C 180,E1 34132.927,E2 34132.927} C_VEL
LIN {X 0,Y 728.632,Z 1120.123,A -85,B 0,C 180,E1 34130.987,E2 34130.987} C_VEL
LIN {X 0,Y 728.422,Z 1133.804,A -85,B 0,C 180,E1 34129.318,E2 34129.318} C_VEL
LIN {X 0,Y 728.29,Z 1145.419,A -85,B 0,C 180,E1 34127.745,E2 34127.745} C_VEL
LIN {X 0,Y 728.151,Z 1156.939,A -85,B 0,C 180,E1 34126.005,E2 34126.005} C_VEL
LIN {X 0,Y 728.047,Z 1169.421,A -85,B 0,C 180,E1 34123.825,E2 34123.825} C_VEL
LIN {X 0,Y 727.973,Z 1178.073,A -85,B 0,C 180,E1 34122.05,E2 34122.05} C_VEL
LIN {X 0,Y 727.953,Z 1185.837,A -85,B 0,C 180,E1 34120.206,E2 34120.206} C_VEL
LIN {X 0,Y 727.927,Z 1193.111,A -85,B 0,C 180,E1 34118.054,E2 34118.054} C_VEL
LIN {X 0,Y 727.914,Z 1198.422,A -85,B 0,C 180,E1 34115.992,E2 34115.992} C_VEL
LIN {X 0,Y 727.907,Z 1202.278,A -85,B 0,C 180,E1 34113.859,E2 34113.859} C_VEL
LIN {X 0,Y 727.908,Z 1204.493,A -85,B 0,C 180,E1 34111.653,E2 34111.653} C_VEL
LIN {X 0,Y 727.89,Z 1204.872,A -85,B 0,C 180,E1 34109.528,E2 34109.528} C_VEL
LIN {X 0,Y 727.906,Z 1203.905,A -85,B 0,C 180,E1 34107.56,E2 34107.56} C_VEL
LIN {X 0,Y 727.908,Z 1201.178,A -85,B 0,C 180,E1 34105.431,E2 34105.431} C_VEL
LIN {X 0,Y 727.916,Z 1196.957,A -85,B 0,C 180,E1 34103.374,E2 34103.374} C_VEL
LIN {X 0,Y 727.936,Z 1191.149,A -85,B 0,C 180,E1 34101.31,E2 34101.31} C_VEL
LIN {X 0,Y 727.944,Z 1183.638,A -85,B 0,C 180,E1 34099.234,E2 34099.234} C_VEL
LIN {X 0,Y 728.028,Z 1173.527,A -85,B 0,C 180,E1 34096.983,E2 34096.983} C_VEL
LIN {X 0,Y 728.084,Z 1164.528,A -85,B 0,C 180,E1 34095.282,E2 34095.282} C_VEL
LIN {X 0,Y 728.168,Z 1154.742,A -85,B 0,C 180,E1 34093.651,E2 34093.651} C_VEL
LIN {X 0,Y 728.298,Z 1144.115,A -85,B 0,C 180,E1 34092.07,E2 34092.07} C_VEL
LIN {X 0,Y 728.489,Z 1130.976,A -85,B 0,C 180,E1 34090.318,E2 34090.318} C_VEL
LIN {X 0,Y 728.74,Z 1113.474,A -85,B 0,C 180,E1 34088.265,E2 34088.265} C_VEL
LIN {X 0,Y 728.955,Z 1098.834,A -85,B 0,C 180,E1 34086.732,E2 34086.732} C_VEL
LIN {X 0,Y 729.277,Z 1082.529,A -85,B 0,C 180,E1 34085.183,E2 34085.183} C_VEL
LIN {X 0,Y 729.687,Z 1061.274,A -85,B 0,C 180,E1 34083.38,E2 34083.38} C_VEL
LIN {X 0,Y 730.038,Z 1043.447,A -85,B 0,C 180,E1 34082.025,E2 34082.025} C_VEL
LIN {X 0,Y 730.495,Z 1023.598,A -85,B 0,C 180,E1 34080.659,E2 34080.659} C_VEL
LIN {X 0,Y 731.013,Z 999.732,A -85,B 0,C 180,E1 34079.204,E2 34079.204} C_VEL
LIN {X 0,Y 731.426,Z 978.536,A -85,B 0,C 180,E1 34078.06,E2 34078.06} C_VEL
LIN {X 0,Y 731.862,Z 957.721,A -85,B 0,C 180,E1 34077.061,E2 34077.061} C_VEL
LIN {X 0,Y 732.438,Z 932.735,A -85,B 0,C 180,E1 34076.013,E2 34076.013} C_VEL
LIN {X 0,Y 732.844,Z 907.027,A -85,B 0,C 180,E1 34075.109,E2 34075.109} C_VEL
LIN {X 0,Y 733.217,Z 883.775,A -85,B 0,C 180,E1 34074.416,E2 34074.416} C_VEL
LIN {X 0,Y 733.575,Z 857.308,A -85,B 0,C 180,E1 34073.785,E2 34073.785} C_VEL
LIN {X 0,Y 733.853,Z 830.107,A -85,B 0,C 180,E1 34073.301,E2 34073.301} C_VEL
LIN {X 0,Y 734.243,Z 746.426,A -85,B 0,C 180,E1 34072.289,E2 34072.289} C_VEL
LIN {X 0,Y 735.141,Z 524.027,A -85,B 0,C 180,E1 34069.603,E2 34069.603} C_VEL
LIN {X 0,Y 735.746,Z 357.454,A -85,B 0,C 180,E1 34067.519,E2 34067.519} C_VEL
LIN {X 0,Y 734.021,Z 349.801,A -85,B 0,C 180,E1 34067.285,E2 34067.285} C_VEL
LIN {X 0,Y 734.688,Z 305.594,A -85,B 0,C 180,E1 34064.677,E2 34064.677} C_VEL
LIN {X 0,Y 734.585,Z 302.1,A -85,B 0,C 180,E1 34064.453,E2 34064.453} C_VEL
LIN {X 0,Y 729.349,Z 291.789,A -85,B 0,C 180,E1 34063.381,E2 34063.381} C_VEL
LIN {X 0,Y 728.174,Z 288.724,A -85,B 0,C 180,E1 34063.036,E2 34063.036} C_VEL
LIN {X 0,Y 728.155,Z 288.528,A -85,B 0,C 180,E1 34060.713,E2 34060.713} C_VEL
LIN {X 0,Y 728.132,Z 288.528,A -85,B 0,C 180,E1 34057.768,E2 34057.768} C_VEL
LIN {X 0,Y 728.142,Z 288.527,A -85,B 0,C 180,E1 34054.934,E2 34054.934} C_VEL
LIN {X 0,Y 728.136,Z 288.522,A -85,B 0,C 180,E1 34052.087,E2 34052.087} C_VEL
LIN {X 0,Y 728.154,Z 288.532,A -85,B 0,C 180,E1 34049.154,E2 34049.154} C_VEL
LIN {X 0,Y 728.149,Z 288.516,A -85,B 0,C 180,E1 34046.099,E2 34046.099} C_VEL
LIN {X 0,Y 728.154,Z 288.526,A -85,B 0,C 180,E1 34043.074,E2 34043.074} C_VEL
LIN {X 0,Y 728.156,Z 288.519,A -85,B 0,C 180,E1 34039.994,E2 34039.994} C_VEL
LIN {X 0,Y 728.154,Z 288.522,A -85,B 0,C 180,E1 34036.925,E2 34036.925} C_VEL
LIN {X 0,Y 728.156,Z 288.519,A -85,B 0,C 180,E1 34033.879,E2 34033.879} C_VEL
LIN {X 0,Y 728.154,Z 288.523,A -85,B 0,C 180,E1 34030.844,E2 34030.844} C_VEL
LIN {X 0,Y 728.153,Z 288.518,A -85,B 0,C 180,E1 34027.813,E2 34027.813} C_VEL
LIN {X 0,Y 728.155,Z 288.53,A -85,B 0,C 180,E1 34024.726,E2 34024.726} C_VEL
LIN {X 0,Y 728.144,Z 288.521,A -85,B 0,C 180,E1 34021.731,E2 34021.731} C_VEL
LIN {X 0,Y 728.155,Z 288.532,A -85,B 0,C 180,E1 34018.741,E2 34018.741} C_VEL
LIN {X 0,Y 728.127,Z 288.525,A -85,B 0,C 180,E1 34015.826,E2 34015.826} C_VEL
LIN {X 0,Y 728.146,Z 288.523,A -85,B 0,C 180,E1 34012.98,E2 34012.98} C_VEL
LIN {X 0,Y 728.13,Z 288.529,A -85,B 0,C 180,E1 34010.116,E2 34010.116} C_VEL
LIN {X 0,Y 728.151,Z 288.52,A -85,B 0,C 180,E1 34007.227,E2 34007.227} C_VEL
LIN {X 0,Y 728.158,Z 288.53,A -85,B 0,C 180,E1 34006.36,E2 34006.36} C_VEL
LIN {X 0,Y 727.162,Z 288.657,A -85,B 0,C 180,E1 34005.754,E2 34005.754} C_VEL
LIN {X 0,Y 720.7,Z 289.455,A -85,B 0,C 180,E1 34004.056,E2 34004.056} C_VEL
LIN {X 0,Y 720.179,Z 289.512,A -85,B 0,C 180,E1 34003.615,E2 34003.615} C_VEL
LIN {X 0,Y 720.214,Z 289.514,A -85,B 0,C 180,E1 34000.739,E2 34000.739} C_VEL
LIN {X 0,Y 720.184,Z 289.518,A -85,B 0,C 180,E1 33997.812,E2 33997.812} C_VEL
LIN {X 0,Y 720.201,Z 289.5,A -85,B 0,C 180,E1 33994.948,E2 33994.948} C_VEL
LIN {X 0,Y 720.195,Z 289.521,A -85,B 0,C 180,E1 33991.833,E2 33991.833} C_VEL
LIN {X 0,Y 720.182,Z 289.503,A -85,B 0,C 180,E1 33988.996,E2 33988.996} C_VEL
LIN {X 0,Y 720.219,Z 289.52,A -85,B 0,C 180,E1 33985.975,E2 33985.975} C_VEL
LIN {X 0,Y 720.167,Z 289.504,A -85,B 0,C 180,E1 33983.145,E2 33983.145} C_VEL
LIN {X 0,Y 720.219,Z 289.514,A -85,B 0,C 180,E1 33980.273,E2 33980.273} C_VEL
LIN {X 0,Y 720.174,Z 289.518,A -85,B 0,C 180,E1 33977.348,E2 33977.348} C_VEL
LIN {X 0,Y 720.176,Z 289.514,A -85,B 0,C 180,E1 33974.628,E2 33974.628} C_VEL
LIN {X 0,Y 720.212,Z 289.522,A -85,B 0,C 180,E1 33971.575,E2 33971.575} C_VEL
LIN {X 0,Y 720.159,Z 289.519,A -85,B 0,C 180,E1 33968.839,E2 33968.839} C_VEL
LIN {X 0,Y 720.212,Z 289.502,A -85,B 0,C 180,E1 33966.06,E2 33966.06} C_VEL
LIN {X 0,Y 720.225,Z 289.699,A -85,B 0,C 180,E1 33964.089,E2 33964.089} C_VEL
LIN {X 0,Y 721.65,Z 293.174,A -85,B 0,C 180,E1 33963.692,E2 33963.692} C_VEL
LIN {X 0,Y 726.483,Z 304.499,A -85,B 0,C 180,E1 33962.557,E2 33962.557} C_VEL
LIN {X 0,Y 725.718,Z 345.772,A -85,B 0,C 180,E1 33959.826,E2 33959.826} C_VEL
LIN {X 0,Y 726.208,Z 348.979,A -85,B 0,C 180,E1 33959.698,E2 33959.698} C_VEL
LIN {X 0,Y 728.084,Z 357.367,A -85,B 0,C 180,E1 33959.476,E2 33959.476} C_VEL
LIN {X 0,Y 726.937,Z 600.768,A -85,B 0,C 180,E1 33956.594,E2 33956.594} C_VEL
LIN {X 0,Y 726.124,Z 779.793,A -85,B 0,C 180,E1 33954.508,E2 33954.508} C_VEL
LIN {X 0,Y 725.885,Z 804.424,A -85,B 0,C 180,E1 33954.102,E2 33954.102} C_VEL
LIN {X 0,Y 725.421,Z 830.035,A -85,B 0,C 180,E1 33953.517,E2 33953.517} C_VEL
LIN {X 0,Y 725.065,Z 851.692,A -85,B 0,C 180,E1 33952.898,E2 33952.898} C_VEL
LIN {X 0,Y 724.623,Z 876.553,A -85,B 0,C 180,E1 33952.044,E2 33952.044} C_VEL
LIN {X 0,Y 724.046,Z 899.793,A -85,B 0,C 180,E1 33951.084,E2 33951.084} C_VEL
LIN {X 0,Y 723.576,Z 919.977,A -85,B 0,C 180,E1 33950.125,E2 33950.125} C_VEL
LIN {X 0,Y 723.041,Z 943.628,A -85,B 0,C 180,E1 33948.838,E2 33948.838} C_VEL
LIN {X 0,Y 722.514,Z 963.354,A -85,B 0,C 180,E1 33947.609,E2 33947.609} C_VEL
LIN {X 0,Y 722.072,Z 983.524,A -85,B 0,C 180,E1 33946.202,E2 33946.202} C_VEL
LIN {X 0,Y 721.609,Z 1002.575,A -85,B 0,C 180,E1 33944.688,E2 33944.688} C_VEL
LIN {X 0,Y 721.227,Z 1019.15,A -85,B 0,C 180,E1 33943.223,E2 33943.223} C_VEL
LIN {X 0,Y 720.871,Z 1037.019,A -85,B 0,C 180,E1 33941.44,E2 33941.44} C_VEL
LIN {X 0,Y 720.61,Z 1050.892,A -85,B 0,C 180,E1 33939.878,E2 33939.878} C_VEL
LIN {X 0,Y 720.391,Z 1065.331,A -85,B 0,C 180,E1 33938.058,E2 33938.058} C_VEL
LIN {X 0,Y 720.216,Z 1077.924,A -85,B 0,C 180,E1 33936.216,E2 33936.216} C_VEL
LIN {X 0,Y 720.099,Z 1087.542,A -85,B 0,C 180,E1 33934.619,E2 33934.619} C_VEL
LIN {X 0,Y 720.019,Z 1096.766,A -85,B 0,C 180,E1 33932.865,E2 33932.865} C_VEL
LIN {X 0,Y 719.949,Z 1105.832,A -85,B 0,C 180,E1 33930.796,E2 33930.796} C_VEL
LIN {X 0,Y 719.935,Z 1112.053,A -85,B 0,C 180,E1 33929.045,E2 33929.045} C_VEL
LIN {X 0,Y 719.919,Z 1116.846,A -85,B 0,C 180,E1 33927.373,E2 33927.373} C_VEL
LIN {X 0,Y 719.894,Z 1121.013,A -85,B 0,C 180,E1 33925.459,E2 33925.459} C_VEL
LIN {X 0,Y 719.9,Z 1123.773,A -85,B 0,C 180,E1 33923.38,E2 33923.38} C_VEL
LIN {X 0,Y 719.913,Z 1124.799,A -85,B 0,C 180,E1 33921.695,E2 33921.695} C_VEL
LIN {X 0,Y 719.897,Z 1124.734,A -85,B 0,C 180,E1 33919.984,E2 33919.984} C_VEL
LIN {X 0,Y 719.908,Z 1123.141,A -85,B 0,C 180,E1 33917.894,E2 33917.894} C_VEL
LIN {X 0,Y 719.898,Z 1120.144,A -85,B 0,C 180,E1 33916.015,E2 33916.015} C_VEL
LIN {X 0,Y 719.919,Z 1116.413,A -85,B 0,C 180,E1 33914.369,E2 33914.369} C_VEL
LIN {X 0,Y 719.931,Z 1111.297,A -85,B 0,C 180,E1 33912.627,E2 33912.627} C_VEL
LIN {X 0,Y 719.99,Z 1103.482,A -85,B 0,C 180,E1 33910.531,E2 33910.531} C_VEL
LIN {X 0,Y 720.018,Z 1095.283,A -85,B 0,C 180,E1 33908.75,E2 33908.75} C_VEL
LIN {X 0,Y 720.123,Z 1086.583,A -85,B 0,C 180,E1 33907.122,E2 33907.122} C_VEL
LIN {X 0,Y 720.281,Z 1074.886,A -85,B 0,C 180,E1 33905.215,E2 33905.215} C_VEL
LIN {X 0,Y 720.444,Z 1061.508,A -85,B 0,C 180,E1 33903.355,E2 33903.355} C_VEL
LIN {X 0,Y 720.663,Z 1048.621,A -85,B 0,C 180,E1 33901.764,E2 33901.764} C_VEL
LIN {X 0,Y 720.981,Z 1031.849,A -85,B 0,C 180,E1 33899.928,E2 33899.928} C_VEL
LIN {X 0,Y 721.302,Z 1016.019,A -85,B 0,C 180,E1 33898.401,E2 33898.401} C_VEL
LIN {X 0,Y 721.739,Z 997.605,A -85,B 0,C 180,E1 33896.802,E2 33896.802} C_VEL
LIN {X 0,Y 722.167,Z 978.092,A -85,B 0,C 180,E1 33895.317,E2 33895.317} C_VEL
LIN {X 0,Y 722.68,Z 958.528,A -85,B 0,C 180,E1 33893.984,E2 33893.984} C_VEL
LIN {X 0,Y 723.189,Z 935.89,A -85,B 0,C 180,E1 33892.631,E2 33892.631} C_VEL
LIN {X 0,Y 723.69,Z 915.432,A -85,B 0,C 180,E1 33891.558,E2 33891.558} C_VEL
LIN {X 0,Y 724.288,Z 891.817,A -85,B 0,C 180,E1 33890.476,E2 33890.476} C_VEL
LIN {X 0,Y 724.737,Z 867.856,A -85,B 0,C 180,E1 33889.552,E2 33889.552} C_VEL
LIN {X 0,Y 725.156,Z 846.092,A -85,B 0,C 180,E1 33888.839,E2 33888.839} C_VEL
LIN {X 0,Y 725.649,Z 819.399,A -85,B 0,C 180,E1 33888.132,E2 33888.132} C_VEL
LIN {X 0,Y 725.926,Z 796.857,A -85,B 0,C 180,E1 33887.672,E2 33887.672} C_VEL
LIN {X 0,Y 726.142,Z 775.915,A -85,B 0,C 180,E1 33887.35,E2 33887.35} C_VEL
LIN {X 0,Y 727.277,Z 526.578,A -85,B 0,C 180,E1 33884.448,E2 33884.448} C_VEL
LIN {X 0,Y 727.927,Z 355.791,A -85,B 0,C 180,E1 33882.405,E2 33882.405} C_VEL
LIN {X 0,Y 725.751,Z 346.783,A -85,B 0,C 180,E1 33882.141,E2 33882.141} C_VEL
LIN {X 0,Y 726.454,Z 305.992,A -85,B 0,C 180,E1 33879.454,E2 33879.454} C_VEL
LIN {X 0,Y 726.25,Z 303.899,A -85,B 0,C 180,E1 33879.296,E2 33879.296} C_VEL
LIN {X 0,Y 720.252,Z 289.825,A -85,B 0,C 180,E1 33877.851,E2 33877.851} C_VEL
LIN {X 0,Y 720.19,Z 289.524,A -85,B 0,C 180,E1 33877.033,E2 33877.033} C_VEL
LIN {X 0,Y 720.214,Z 289.519,A -85,B 0,C 180,E1 33874.166,E2 33874.166} C_VEL
LIN {X 0,Y 720.207,Z 289.514,A -85,B 0,C 180,E1 33871.188,E2 33871.188} C_VEL
LIN {X 0,Y 720.223,Z 289.518,A -85,B 0,C 180,E1 33868.166,E2 33868.166} C_VEL
LIN {X 0,Y 720.208,Z 289.507,A -85,B 0,C 180,E1 33865.052,E2 33865.052} C_VEL
LIN {X 0,Y 720.219,Z 289.51,A -85,B 0,C 180,E1 33862.015,E2 33862.015} C_VEL
LIN {X 0,Y 720.215,Z 289.511,A -85,B 0,C 180,E1 33858.958,E2 33858.958} C_VEL
LIN {X 0,Y 720.219,Z 289.513,A -85,B 0,C 180,E1 33855.873,E2 33855.873} C_VEL
LIN {X 0,Y 720.213,Z 289.504,A -85,B 0,C 180,E1 33852.753,E2 33852.753} C_VEL
LIN {X 0,Y 720.216,Z 289.522,A -85,B 0,C 180,E1 33849.671,E2 33849.671} C_VEL
LIN {X 0,Y 720.215,Z 289.499,A -85,B 0,C 180,E1 33846.617,E2 33846.617} C_VEL
LIN {X 0,Y 720.217,Z 289.519,A -85,B 0,C 180,E1 33843.582,E2 33843.582} C_VEL
LIN {X 0,Y 720.22,Z 289.504,A -85,B 0,C 180,E1 33840.477,E2 33840.477} C_VEL
LIN {X 0,Y 720.213,Z 289.513,A -85,B 0,C 180,E1 33837.374,E2 33837.374} C_VEL
LIN {X 0,Y 720.217,Z 289.508,A -85,B 0,C 180,E1 33834.343,E2 33834.343} C_VEL
LIN {X 0,Y 720.216,Z 289.51,A -85,B 0,C 180,E1 33831.284,E2 33831.284} C_VEL
LIN {X 0,Y 720.218,Z 289.51,A -85,B 0,C 180,E1 33828.224,E2 33828.224} C_VEL
LIN {X 0,Y 720.219,Z 289.509,A -85,B 0,C 180,E1 33825.117,E2 33825.117} C_VEL
LIN {X 0,Y 720.215,Z 289.51,A -85,B 0,C 180,E1 33822.049,E2 33822.049} C_VEL
LIN {X 0,Y 720.214,Z 289.517,A -85,B 0,C 180,E1 33818.926,E2 33818.926} C_VEL
LIN {X 0,Y 720.213,Z 289.502,A -85,B 0,C 180,E1 33815.91,E2 33815.91} C_VEL
LIN {X 0,Y 720.216,Z 289.518,A -85,B 0,C 180,E1 33812.822,E2 33812.822} C_VEL
LIN {X 0,Y 720.216,Z 289.511,A -85,B 0,C 180,E1 33809.737,E2 33809.737} C_VEL
LIN {X 0,Y 720.214,Z 289.52,A -85,B 0,C 180,E1 33806.648,E2 33806.648} C_VEL
LIN {X 0,Y 720.207,Z 289.515,A -85,B 0,C 180,E1 33803.63,E2 33803.63} C_VEL
LIN {X 0,Y 720.214,Z 289.509,A -85,B 0,C 180,E1 33800.517,E2 33800.517} C_VEL
LIN {X 0,Y 720.219,Z 289.666,A -85,B 0,C 180,E1 33797.609,E2 33797.609} C_VEL
LIN {X 0,Y 720.468,Z 290.736,A -85,B 0,C 180,E1 33797.444,E2 33797.444} C_VEL
LIN {X 0,Y 728.471,Z 306.646,A -85,B 0,C 180,E1 33795.754,E2 33795.754} C_VEL
LIN {X 0,Y 727.641,Z 349.819,A -85,B 0,C 180,E1 33793.181,E2 33793.181} C_VEL
LIN {X 0,Y 729.931,Z 360.759,A -85,B 0,C 180,E1 33792.857,E2 33792.857} C_VEL
LIN {X 0,Y 728.784,Z 572.111,A -85,B 0,C 180,E1 33790.213,E2 33790.213} C_VEL
LIN {X 0,Y 727.663,Z 797.321,A -85,B 0,C 180,E1 33787.49,E2 33787.49} C_VEL
LIN {X 0,Y 727.39,Z 834.846,A -85,B 0,C 180,E1 33787.006,E2 33787.006} C_VEL
LIN {X 0,Y 726.983,Z 862.203,A -85,B 0,C 180,E1 33786.486,E2 33786.486} C_VEL
LIN {X 0,Y 726.551,Z 887.845,A -85,B 0,C 180,E1 33785.846,E2 33785.846} C_VEL
LIN {X 0,Y 725.974,Z 916.207,A -85,B 0,C 180,E1 33784.956,E2 33784.956} C_VEL
LIN {X 0,Y 725.376,Z 939.91,A -85,B 0,C 180,E1 33784.06,E2 33784.06} C_VEL
LIN {X 0,Y 724.837,Z 961.081,A -85,B 0,C 180,E1 33783.139,E2 33783.139} C_VEL
LIN {X 0,Y 724.299,Z 983.238,A -85,B 0,C 180,E1 33782.045,E2 33782.045} C_VEL
LIN {X 0,Y 723.607,Z 1008.624,A -85,B 0,C 180,E1 33780.609,E2 33780.609} C_VEL
LIN {X 0,Y 723.047,Z 1028.237,A -85,B 0,C 180,E1 33779.355,E2 33779.355} C_VEL
LIN {X 0,Y 722.54,Z 1047.294,A -85,B 0,C 180,E1 33778.005,E2 33778.005} C_VEL
LIN {X 0,Y 721.988,Z 1069.758,A -85,B 0,C 180,E1 33776.217,E2 33776.217} C_VEL
LIN {X 0,Y 721.544,Z 1086.384,A -85,B 0,C 180,E1 33774.739,E2 33774.739} C_VEL
LIN {X 0,Y 721.208,Z 1103.096,A -85,B 0,C 180,E1 33773.1,E2 33773.1} C_VEL
LIN {X 0,Y 720.819,Z 1120.836,A -85,B 0,C 180,E1 33771.14,E2 33771.14} C_VEL
LIN {X 0,Y 720.583,Z 1133.806,A -85,B 0,C 180,E1 33769.536,E2 33769.536} C_VEL
LIN {X 0,Y 720.388,Z 1146.003,A -85,B 0,C 180,E1 33767.863,E2 33767.863} C_VEL
LIN {X 0,Y 720.214,Z 1158.902,A -85,B 0,C 180,E1 33765.872,E2 33765.872} C_VEL
LIN {X 0,Y 720.078,Z 1170.244,A -85,B 0,C 180,E1 33763.817,E2 33763.817} C_VEL
LIN {X 0,Y 719.995,Z 1178.432,A -85,B 0,C 180,E1 33762.104,E2 33762.104} C_VEL
LIN {X 0,Y 719.965,Z 1186.134,A -85,B 0,C 180,E1 33760.239,E2 33760.239} C_VEL
LIN {X 0,Y 719.933,Z 1193.546,A -85,B 0,C 180,E1 33758,E2 33758} C_VEL
LIN {X 0,Y 719.918,Z 1198.937,A -85,B 0,C 180,E1 33755.819,E2 33755.819} C_VEL
LIN {X 0,Y 719.909,Z 1202.484,A -85,B 0,C 180,E1 33753.743,E2 33753.743} C_VEL
LIN {X 0,Y 719.909,Z 1204.549,A -85,B 0,C 180,E1 33751.592,E2 33751.592} C_VEL
LIN {X 0,Y 719.89,Z 1204.872,A -85,B 0,C 180,E1 33749.523,E2 33749.523} C_VEL
LIN {X 0,Y 719.906,Z 1203.902,A -85,B 0,C 180,E1 33747.532,E2 33747.532} C_VEL
LIN {X 0,Y 719.907,Z 1201.178,A -85,B 0,C 180,E1 33745.38,E2 33745.38} C_VEL
LIN {X 0,Y 719.917,Z 1196.832,A -85,B 0,C 180,E1 33743.249,E2 33743.249} C_VEL
LIN {X 0,Y 719.937,Z 1190.891,A -85,B 0,C 180,E1 33741.132,E2 33741.132} C_VEL
LIN {X 0,Y 719.972,Z 1183.001,A -85,B 0,C 180,E1 33738.951,E2 33738.951} C_VEL
LIN {X 0,Y 720.061,Z 1173.152,A -85,B 0,C 180,E1 33736.762,E2 33736.762} C_VEL
LIN {X 0,Y 720.128,Z 1164.064,A -85,B 0,C 180,E1 33735.034,E2 33735.034} C_VEL
LIN {X 0,Y 720.263,Z 1154.221,A -85,B 0,C 180,E1 33733.383,E2 33733.383} C_VEL
LIN {X 0,Y 720.441,Z 1142.511,A -85,B 0,C 180,E1 33731.637,E2 33731.637} C_VEL
LIN {X 0,Y 720.722,Z 1126.521,A -85,B 0,C 180,E1 33729.537,E2 33729.537} C_VEL
LIN {X 0,Y 720.991,Z 1111.843,A -85,B 0,C 180,E1 33727.839,E2 33727.839} C_VEL
LIN {X 0,Y 721.307,Z 1097.128,A -85,B 0,C 180,E1 33726.297,E2 33726.297} C_VEL
LIN {X 0,Y 721.784,Z 1077.881,A -85,B 0,C 180,E1 33724.481,E2 33724.481} C_VEL
LIN {X 0,Y 722.23,Z 1059.06,A -85,B 0,C 180,E1 33722.905,E2 33722.905} C_VEL
LIN {X 0,Y 722.736,Z 1041.03,A -85,B 0,C 180,E1 33721.537,E2 33721.537} C_VEL
LIN {X 0,Y 723.365,Z 1018.082,A -85,B 0,C 180,E1 33719.976,E2 33719.976} C_VEL
LIN {X 0,Y 723.901,Z 996.241,A -85,B 0,C 180,E1 33718.666,E2 33718.666} C_VEL
LIN {X 0,Y 724.473,Z 975.869,A -85,B 0,C 180,E1 33717.576,E2 33717.576} C_VEL
LIN {X 0,Y 725.163,Z 951.713,A -85,B 0,C 180,E1 33716.434,E2 33716.434} C_VEL
LIN {X 0,Y 725.714,Z 926.414,A -85,B 0,C 180,E1 33715.415,E2 33715.415} C_VEL
LIN {X 0,Y 726.174,Z 904.862,A -85,B 0,C 180,E1 33714.67,E2 33714.67} C_VEL
LIN {X 0,Y 726.647,Z 881.764,A -85,B 0,C 180,E1 33713.988,E2 33713.988} C_VEL
LIN {X 0,Y 727.127,Z 854.691,A -85,B 0,C 180,E1 33713.354,E2 33713.354} C_VEL
LIN {X 0,Y 727.448,Z 827.378,A -85,B 0,C 180,E1 33712.882,E2 33712.882} C_VEL
LIN {X 0,Y 728.665,Z 593.854,A -85,B 0,C 180,E1 33710.053,E2 33710.053} C_VEL
LIN {X 0,Y 729.828,Z 379.687,A -85,B 0,C 180,E1 33707.384,E2 33707.384} C_VEL
LIN {X 0,Y 729.777,Z 359.234,A -85,B 0,C 180,E1 33707.112,E2 33707.112} C_VEL
LIN {X 0,Y 727.642,Z 349.823,A -85,B 0,C 180,E1 33706.819,E2 33706.819} C_VEL
LIN {X 0,Y 728.467,Z 306.594,A -85,B 0,C 180,E1 33704.243,E2 33704.243} C_VEL
LIN {X 0,Y 721.854,Z 293.417,A -85,B 0,C 180,E1 33702.853,E2 33702.853} C_VEL
LIN {X 0,Y 720.237,Z 289.76,A -85,B 0,C 180,E1 33702.434,E2 33702.434} C_VEL
LIN {X 0,Y 720.218,Z 289.502,A -85,B 0,C 180,E1 33701.47,E2 33701.47} C_VEL
LIN {X 0,Y 720.214,Z 289.508,A -85,B 0,C 180,E1 33698.46,E2 33698.46} C_VEL
LIN {X 0,Y 720.22,Z 289.521,A -85,B 0,C 180,E1 33695.375,E2 33695.375} C_VEL
LIN {X 0,Y 720.212,Z 289.508,A -85,B 0,C 180,E1 33692.279,E2 33692.279} C_VEL
LIN {X 0,Y 720.219,Z 289.521,A -85,B 0,C 180,E1 33689.254,E2 33689.254} C_VEL
LIN {X 0,Y 720.214,Z 289.503,A -85,B 0,C 180,E1 33686.199,E2 33686.199} C_VEL
LIN {X 0,Y 720.216,Z 289.515,A -85,B 0,C 180,E1 33683.135,E2 33683.135} C_VEL
LIN {X 0,Y 720.217,Z 289.507,A -85,B 0,C 180,E1 33680.055,E2 33680.055} C_VEL
LIN {X 0,Y 720.215,Z 289.509,A -85,B 0,C 180,E1 33676.951,E2 33676.951} C_VEL
LIN {X 0,Y 720.217,Z 289.508,A -85,B 0,C 180,E1 33673.897,E2 33673.897} C_VEL
LIN {X 0,Y 720.213,Z 289.509,A -85,B 0,C 180,E1 33670.803,E2 33670.803} C_VEL
LIN {X 0,Y 720.217,Z 289.506,A -85,B 0,C 180,E1 33667.739,E2 33667.739} C_VEL
LIN {X 0,Y 720.21,Z 289.519,A -85,B 0,C 180,E1 33664.619,E2 33664.619} C_VEL
LIN {X 0,Y 720.216,Z 289.508,A -85,B 0,C 180,E1 33661.591,E2 33661.591} C_VEL
LIN {X 0,Y 720.21,Z 289.518,A -85,B 0,C 180,E1 33658.488,E2 33658.488} C_VEL
LIN {X 0,Y 720.214,Z 289.51,A -85,B 0,C 180,E1 33655.461,E2 33655.461} C_VEL
LIN {X 0,Y 720.207,Z 289.521,A -85,B 0,C 180,E1 33652.341,E2 33652.341} C_VEL
LIN {X 0,Y 720.206,Z 289.51,A -85,B 0,C 180,E1 33649.359,E2 33649.359} C_VEL
LIN {X 0,Y 720.212,Z 289.52,A -85,B 0,C 180,E1 33646.267,E2 33646.267} C_VEL
LIN {X 0,Y 720.179,Z 289.512,A -85,B 0,C 180,E1 33643.615,E2 33643.615} C_VEL
LIN {X 0,Y 719.215,Z 289.635,A -85,B 0,C 180,E1 33643.002,E2 33643.002} C_VEL
LIN {X 0,Y 712.815,Z 290.434,A -85,B 0,C 180,E1 33641.286,E2 33641.286} C_VEL
LIN {X 0,Y 712.278,Z 290.501,A -85,B 0,C 180,E1 33640.839,E2 33640.839} C_VEL
LIN {X 0,Y 712.252,Z 290.508,A -85,B 0,C 180,E1 33637.896,E2 33637.896} C_VEL
LIN {X 0,Y 712.257,Z 290.487,A -85,B 0,C 180,E1 33635.004,E2 33635.004} C_VEL
LIN {X 0,Y 712.259,Z 290.51,A -85,B 0,C 180,E1 33631.856,E2 33631.856} C_VEL
LIN {X 0,Y 712.243,Z 290.491,A -85,B 0,C 180,E1 33628.988,E2 33628.988} C_VEL
LIN {X 0,Y 712.277,Z 290.511,A -85,B 0,C 180,E1 33625.915,E2 33625.915} C_VEL
LIN {X 0,Y 712.229,Z 290.49,A -85,B 0,C 180,E1 33623.068,E2 33623.068} C_VEL
LIN {X 0,Y 712.28,Z 290.506,A -85,B 0,C 180,E1 33620.161,E2 33620.161} C_VEL
LIN {X 0,Y 712.23,Z 290.506,A -85,B 0,C 180,E1 33617.24,E2 33617.24} C_VEL
LIN {X 0,Y 712.252,Z 290.502,A -85,B 0,C 180,E1 33614.467,E2 33614.467} C_VEL
LIN {X 0,Y 712.242,Z 290.509,A -85,B 0,C 180,E1 33611.317,E2 33611.317} C_VEL
LIN {X 0,Y 712.223,Z 290.507,A -85,B 0,C 180,E1 33608.661,E2 33608.661} C_VEL
LIN {X 0,Y 712.28,Z 290.488,A -85,B 0,C 180,E1 33605.768,E2 33605.768} C_VEL
LIN {X 0,Y 712.26,Z 290.8,A -85,B 0,C 180,E1 33604.599,E2 33604.599} C_VEL
LIN {X 0,Y 714.843,Z 297.007,A -85,B 0,C 180,E1 33603.923,E2 33603.923} C_VEL
LIN {X 0,Y 719.79,Z 308.386,A -85,B 0,C 180,E1 33602.76,E2 33602.76} C_VEL
LIN {X 0,Y 719.004,Z 346.796,A -85,B 0,C 180,E1 33600.202,E2 33600.202} C_VEL
LIN {X 0,Y 721.806,Z 359.299,A -85,B 0,C 180,E1 33599.85,E2 33599.85} C_VEL
LIN {X 0,Y 720.411,Z 604.116,A -85,B 0,C 180,E1 33596.926,E2 33596.926} C_VEL
LIN {X 0,Y 719.442,Z 780.033,A -85,B 0,C 180,E1 33594.858,E2 33594.858} C_VEL
LIN {X 0,Y 719.137,Z 805.302,A -85,B 0,C 180,E1 33594.436,E2 33594.436} C_VEL
LIN {X 0,Y 718.595,Z 830.516,A -85,B 0,C 180,E1 33593.852,E2 33593.852} C_VEL
LIN {X 0,Y 718.165,Z 851.981,A -85,B 0,C 180,E1 33593.232,E2 33593.232} C_VEL
LIN {X 0,Y 717.613,Z 877.153,A -85,B 0,C 180,E1 33592.357,E2 33592.357} C_VEL
LIN {X 0,Y 716.944,Z 900.337,A -85,B 0,C 180,E1 33591.388,E2 33591.388} C_VEL
LIN {X 0,Y 716.349,Z 921.31,A -85,B 0,C 180,E1 33590.38,E2 33590.38} C_VEL
LIN {X 0,Y 715.667,Z 945.427,A -85,B 0,C 180,E1 33589.04,E2 33589.04} C_VEL
LIN {X 0,Y 715.069,Z 964.501,A -85,B 0,C 180,E1 33587.832,E2 33587.832} C_VEL
LIN {X 0,Y 714.496,Z 985.497,A -85,B 0,C 180,E1 33586.336,E2 33586.336} C_VEL
LIN {X 0,Y 713.958,Z 1003.836,A -85,B 0,C 180,E1 33584.849,E2 33584.849} C_VEL
LIN {X 0,Y 713.492,Z 1021.185,A -85,B 0,C 180,E1 33583.287,E2 33583.287} C_VEL
LIN {X 0,Y 713.071,Z 1037.995,A -85,B 0,C 180,E1 33581.567,E2 33581.567} C_VEL
LIN {X 0,Y 712.759,Z 1051.671,A -85,B 0,C 180,E1 33580.002,E2 33580.002} C_VEL
LIN {X 0,Y 712.491,Z 1066.086,A -85,B 0,C 180,E1 33578.148,E2 33578.148} C_VEL
LIN {X 0,Y 712.282,Z 1078.58,A -85,B 0,C 180,E1 33576.286,E2 33576.286} C_VEL
LIN {X 0,Y 712.138,Z 1088.578,A -85,B 0,C 180,E1 33574.59,E2 33574.59} C_VEL
LIN {X 0,Y 712.049,Z 1098.797,A -85,B 0,C 180,E1 33572.575,E2 33572.575} C_VEL
LIN {X 0,Y 711.953,Z 1106.517,A -85,B 0,C 180,E1 33570.724,E2 33570.724} C_VEL
LIN {X 0,Y 711.94,Z 1112.375,A -85,B 0,C 180,E1 33569.034,E2 33569.034} C_VEL
LIN {X 0,Y 711.919,Z 1117.107,A -85,B 0,C 180,E1 33567.344,E2 33567.344} C_VEL
LIN {X 0,Y 711.895,Z 1121.465,A -85,B 0,C 180,E1 33565.247,E2 33565.247} C_VEL
LIN {X 0,Y 711.895,Z 1123.858,A -85,B 0,C 180,E1 33563.306,E2 33563.306} C_VEL
LIN {X 0,Y 711.907,Z 1124.827,A -85,B 0,C 180,E1 33561.601,E2 33561.601} C_VEL
LIN {X 0,Y 711.91,Z 1124.665,A -85,B 0,C 180,E1 33559.725,E2 33559.725} C_VEL
LIN {X 0,Y 711.915,Z 1122.766,A -85,B 0,C 180,E1 33557.591,E2 33557.591} C_VEL
LIN {X 0,Y 711.913,Z 1119.938,A -85,B 0,C 180,E1 33555.855,E2 33555.855} C_VEL
LIN {X 0,Y 711.91,Z 1115.93,A -85,B 0,C 180,E1 33554.105,E2 33554.105} C_VEL
LIN {X 0,Y 711.949,Z 1109.882,A -85,B 0,C 180,E1 33552.088,E2 33552.088} C_VEL
LIN {X 0,Y 711.993,Z 1102.265,A -85,B 0,C 180,E1 33550.133,E2 33550.133} C_VEL
LIN {X 0,Y 712.059,Z 1094.735,A -85,B 0,C 180,E1 33548.501,E2 33548.501} C_VEL
LIN {X 0,Y 712.19,Z 1085.466,A -85,B 0,C 180,E1 33546.765,E2 33546.765} C_VEL
LIN {X 0,Y 712.384,Z 1072.275,A -85,B 0,C 180,E1 33544.654,E2 33544.654} C_VEL
LIN {X 0,Y 712.61,Z 1060.032,A -85,B 0,C 180,E1 33542.961,E2 33542.961} C_VEL
LIN {X 0,Y 712.929,Z 1045.359,A -85,B 0,C 180,E1 33541.155,E2 33541.155} C_VEL
LIN {X 0,Y 713.282,Z 1028.966,A -85,B 0,C 180,E1 33539.398,E2 33539.398} C_VEL
LIN {X 0,Y 713.705,Z 1013.283,A -85,B 0,C 180,E1 33537.891,E2 33537.891} C_VEL
LIN {X 0,Y 714.242,Z 993.32,A -85,B 0,C 180,E1 33536.189,E2 33536.189} C_VEL
LIN {X 0,Y 714.779,Z 975.056,A -85,B 0,C 180,E1 33534.808,E2 33534.808} C_VEL
LIN {X 0,Y 715.438,Z 951.89,A -85,B 0,C 180,E1 33533.262,E2 33533.262} C_VEL
LIN {X 0,Y 716.059,Z 931.768,A -85,B 0,C 180,E1 33532.088,E2 33532.088} C_VEL
LIN {X 0,Y 716.758,Z 908.886,A -85,B 0,C 180,E1 33530.911,E2 33530.911} C_VEL
LIN {X 0,Y 717.346,Z 884.89,A -85,B 0,C 180,E1 33529.861,E2 33529.861} C_VEL
LIN {X 0,Y 717.913,Z 863.526,A -85,B 0,C 180,E1 33529.059,E2 33529.059} C_VEL
LIN {X 0,Y 718.522,Z 837.706,A -85,B 0,C 180,E1 33528.252,E2 33528.252} C_VEL
LIN {X 0,Y 718.917,Z 814.6,A -85,B 0,C 180,E1 33527.675,E2 33527.675} C_VEL
LIN {X 0,Y 719.24,Z 792.495,A -85,B 0,C 180,E1 33527.241,E2 33527.241} C_VEL
LIN {X 0,Y 719.589,Z 761.61,A -85,B 0,C 180,E1 33526.818,E2 33526.818} C_VEL
LIN {X 0,Y 720.884,Z 518.365,A -85,B 0,C 180,E1 33523.97,E2 33523.97} C_VEL
LIN {X 0,Y 721.646,Z 357.724,A -85,B 0,C 180,E1 33522.03,E2 33522.03} C_VEL
LIN {X 0,Y 718.98,Z 346.409,A -85,B 0,C 180,E1 33521.687,E2 33521.687} C_VEL
LIN {X 0,Y 719.792,Z 308.27,A -85,B 0,C 180,E1 33519.142,E2 33519.142} C_VEL
LIN {X 0,Y 713.123,Z 293.208,A -85,B 0,C 180,E1 33517.584,E2 33517.584} C_VEL
LIN {X 0,Y 712.282,Z 290.659,A -85,B 0,C 180,E1 33517.277,E2 33517.277} C_VEL
LIN {X 0,Y 712.277,Z 290.509,A -85,B 0,C 180,E1 33514.356,E2 33514.356} C_VEL
LIN {X 0,Y 712.274,Z 290.503,A -85,B 0,C 180,E1 33511.253,E2 33511.253} C_VEL
LIN {X 0,Y 712.285,Z 290.506,A -85,B 0,C 180,E1 33508.171,E2 33508.171} C_VEL
LIN {X 0,Y 712.272,Z 290.495,A -85,B 0,C 180,E1 33505.084,E2 33505.084} C_VEL
LIN {X 0,Y 712.281,Z 290.496,A -85,B 0,C 180,E1 33502.013,E2 33502.013} C_VEL
LIN {X 0,Y 712.273,Z 290.501,A -85,B 0,C 180,E1 33498.892,E2 33498.892} C_VEL
LIN {X 0,Y 712.279,Z 290.5,A -85,B 0,C 180,E1 33495.887,E2 33495.887} C_VEL
LIN {X 0,Y 712.277,Z 290.492,A -85,B 0,C 180,E1 33492.815,E2 33492.815} C_VEL
LIN {X 0,Y 712.279,Z 290.511,A -85,B 0,C 180,E1 33489.698,E2 33489.698} C_VEL
LIN {X 0,Y 712.275,Z 290.487,A -85,B 0,C 180,E1 33486.61,E2 33486.61} C_VEL
LIN {X 0,Y 712.276,Z 290.507,A -85,B 0,C 180,E1 33483.541,E2 33483.541} C_VEL
LIN {X 0,Y 712.281,Z 290.492,A -85,B 0,C 180,E1 33480.483,E2 33480.483} C_VEL
LIN {X 0,Y 712.276,Z 290.501,A -85,B 0,C 180,E1 33477.425,E2 33477.425} C_VEL
LIN {X 0,Y 712.278,Z 290.497,A -85,B 0,C 180,E1 33474.361,E2 33474.361} C_VEL
LIN {X 0,Y 712.277,Z 290.496,A -85,B 0,C 180,E1 33471.28,E2 33471.28} C_VEL
LIN {X 0,Y 712.28,Z 290.499,A -85,B 0,C 180,E1 33468.173,E2 33468.173} C_VEL
LIN {X 0,Y 712.279,Z 290.496,A -85,B 0,C 180,E1 33465.114,E2 33465.114} C_VEL
LIN {X 0,Y 712.277,Z 290.499,A -85,B 0,C 180,E1 33462.011,E2 33462.011} C_VEL
LIN {X 0,Y 712.275,Z 290.504,A -85,B 0,C 180,E1 33458.938,E2 33458.938} C_VEL
LIN {X 0,Y 712.278,Z 290.489,A -85,B 0,C 180,E1 33455.844,E2 33455.844} C_VEL
LIN {X 0,Y 712.273,Z 290.505,A -85,B 0,C 180,E1 33452.765,E2 33452.765} C_VEL
LIN {X 0,Y 712.28,Z 290.5,A -85,B 0,C 180,E1 33449.689,E2 33449.689} C_VEL
LIN {X 0,Y 712.273,Z 290.508,A -85,B 0,C 180,E1 33446.613,E2 33446.613} C_VEL
LIN {X 0,Y 712.273,Z 290.504,A -85,B 0,C 180,E1 33443.548,E2 33443.548} C_VEL
LIN {X 0,Y 712.268,Z 290.497,A -85,B 0,C 180,E1 33440.414,E2 33440.414} C_VEL
LIN {X 0,Y 712.285,Z 290.707,A -85,B 0,C 180,E1 33438.21,E2 33438.21} C_VEL
LIN {X 0,Y 713.539,Z 293.925,A -85,B 0,C 180,E1 33437.838,E2 33437.838} C_VEL
LIN {X 0,Y 715.05,Z 296.802,A -85,B 0,C 180,E1 33437.514,E2 33437.514} C_VEL
LIN {X 0,Y 722.21,Z 311.062,A -85,B 0,C 180,E1 33435.985,E2 33435.985} C_VEL
LIN {X 0,Y 721.32,Z 349.992,A -85,B 0,C 180,E1 33433.648,E2 33433.648} C_VEL
LIN {X 0,Y 724.042,Z 362.68,A -85,B 0,C 180,E1 33433.265,E2 33433.265} C_VEL
LIN {X 0,Y 722.654,Z 573.817,A -85,B 0,C 180,E1 33430.603,E2 33430.603} C_VEL
LIN {X 0,Y 721.298,Z 798.975,A -85,B 0,C 180,E1 33427.859,E2 33427.859} C_VEL
LIN {X 0,Y 720.972,Z 835.283,A -85,B 0,C 180,E1 33427.384,E2 33427.384} C_VEL
LIN {X 0,Y 720.48,Z 862.704,A -85,B 0,C 180,E1 33426.857,E2 33426.857} C_VEL
LIN {X 0,Y 719.968,Z 888.124,A -85,B 0,C 180,E1 33426.217,E2 33426.217} C_VEL
LIN {X 0,Y 719.266,Z 916.702,A -85,B 0,C 180,E1 33425.311,E2 33425.311} C_VEL
LIN {X 0,Y 718.599,Z 939.498,A -85,B 0,C 180,E1 33424.444,E2 33424.444} C_VEL
LIN {X 0,Y 717.94,Z 960.704,A -85,B 0,C 180,E1 33423.518,E2 33423.518} C_VEL
LIN {X 0,Y 717.251,Z 982.992,A -85,B 0,C 180,E1 33422.412,E2 33422.412} C_VEL
LIN {X 0,Y 716.464,Z 1007.891,A -85,B 0,C 180,E1 33420.995,E2 33420.995} C_VEL
LIN {X 0,Y 715.786,Z 1027.576,A -85,B 0,C 180,E1 33419.728,E2 33419.728} C_VEL
LIN {X 0,Y 715.191,Z 1045.811,A -85,B 0,C 180,E1 33418.431,E2 33418.431} C_VEL
LIN {X 0,Y 714.548,Z 1067.219,A -85,B 0,C 180,E1 33416.735,E2 33416.735} C_VEL
LIN {X 0,Y 713.972,Z 1085.453,A -85,B 0,C 180,E1 33415.108,E2 33415.108} C_VEL
LIN {X 0,Y 713.509,Z 1101.396,A -85,B 0,C 180,E1 33413.539,E2 33413.539} C_VEL
LIN {X 0,Y 713.048,Z 1120.127,A -85,B 0,C 180,E1 33411.468,E2 33411.468} C_VEL
LIN {X 0,Y 712.742,Z 1134.091,A -85,B 0,C 180,E1 33409.723,E2 33409.723} C_VEL
LIN {X 0,Y 712.498,Z 1146.005,A -85,B 0,C 180,E1 33408.067,E2 33408.067} C_VEL
LIN {X 0,Y 712.28,Z 1158.901,A -85,B 0,C 180,E1 33406.054,E2 33406.054} C_VEL
LIN {X 0,Y 712.124,Z 1170.245,A -85,B 0,C 180,E1 33403.975,E2 33403.975} C_VEL
LIN {X 0,Y 712.027,Z 1178.433,A -85,B 0,C 180,E1 33402.242,E2 33402.242} C_VEL
LIN {X 0,Y 711.979,Z 1186.134,A -85,B 0,C 180,E1 33400.356,E2 33400.356} C_VEL
LIN {X 0,Y 711.935,Z 1193.355,A -85,B 0,C 180,E1 33398.155,E2 33398.155} C_VEL
LIN {X 0,Y 711.916,Z 1198.765,A -85,B 0,C 180,E1 33395.966,E2 33395.966} C_VEL
LIN {X 0,Y 711.907,Z 1202.382,A -85,B 0,C 180,E1 33393.866,E2 33393.866} C_VEL
LIN {X 0,Y 711.909,Z 1204.549,A -85,B 0,C 180,E1 33391.61,E2 33391.61} C_VEL
LIN {X 0,Y 711.89,Z 1204.872,A -85,B 0,C 180,E1 33389.517,E2 33389.517} C_VEL
LIN {X 0,Y 711.907,Z 1203.967,A -85,B 0,C 180,E1 33387.585,E2 33387.585} C_VEL
LIN {X 0,Y 711.908,Z 1201.303,A -85,B 0,C 180,E1 33385.408,E2 33385.408} C_VEL
LIN {X 0,Y 711.919,Z 1197.152,A -85,B 0,C 180,E1 33383.306,E2 33383.306} C_VEL
LIN {X 0,Y 711.945,Z 1191.397,A -85,B 0,C 180,E1 33381.195,E2 33381.195} C_VEL
